LIN {X 0,Y 133.458,Z 310.494,A -85,B 0,C 180,E1 -25964.008,E2 -25964.008} C_VEL
LIN {X 0,Y 138.592,Z 326.058,A -85,B 0,C 180,E1 -25966.491,E2 -25966.491} C_VEL
LIN {X 0,Y 134.753,Z 373.673,A -85,B 0,C 180,E1 -25969.183,E2 -25969.183} C_VEL
LIN {X 0,Y 132.897,Z 387.385,A -85,B 0,C 180,E1 -25970.481,E2 -25970.481} C_VEL
LIN {X 0,Y 130.585,Z 400,A -85,B 0,C 180,E1 -25972.246,E2 -25972.246} C_VEL
LIN {X 0,Y 127.54,Z 412.416,A -85,B 0,C 180,E1 -25974.642,E2 -25974.642} C_VEL
LIN {X 0,Y 124.46,Z 423.666,A -85,B 0,C 180,E1 -25977.554,E2 -25977.554} C_VEL
LIN {X 0,Y 121.733,Z 432.92,A -85,B 0,C 180,E1 -25980.641,E2 -25980.641} C_VEL
LIN {X 0,Y 118.797,Z 442.262,A -85,B 0,C 180,E1 -25984.596,E2 -25984.596} C_VEL
LIN {X 0,Y 115.975,Z 451.38,A -85,B 0,C 180,E1 -25989.602,E2 -25989.602} C_VEL
LIN {X 0,Y 113.968,Z 458.709,A -85,B 0,C 180,E1 -25994.8,E2 -25994.8} C_VEL
LIN {X 0,Y 112.959,Z 463.637,A -85,B 0,C 180,E1 -25999.236,E2 -25999.236} C_VEL
LIN {X 0,Y 112.321,Z 468.377,A -85,B 0,C 180,E1 -26004.608,E2 -26004.608} C_VEL
LIN {X 0,Y 112.287,Z 471.952,A -85,B 0,C 180,E1 -26009.994,E2 -26009.994} C_VEL
LIN {X 0,Y 112.224,Z 473.743,A -85,B 0,C 180,E1 -26013.584,E2 -26013.584} C_VEL
LIN {X 0,Y 112.956,Z 476.023,A -85,B 0,C 180,E1 -26020.751,E2 -26020.751} C_VEL
LIN {X 0,Y 115.182,Z 476.815,A -85,B 0,C 180,E1 -26027.757,E2 -26027.757} C_VEL
LIN {X 0,Y 116.858,Z 476.66,A -85,B 0,C 180,E1 -26031.146,E2 -26031.146} C_VEL
LIN {X 0,Y 121.585,Z 475.187,A -85,B 0,C 180,E1 -26037.537,E2 -26037.537} C_VEL
LIN {X 0,Y 127.888,Z 472.229,A -85,B 0,C 180,E1 -26043.329,E2 -26043.329} C_VEL
LIN {X 0,Y 133.433,Z 468.921,A -85,B 0,C 180,E1 -26047.273,E2 -26047.273} C_VEL
LIN {X 0,Y 139.39,Z 464.647,A -85,B 0,C 180,E1 -26050.947,E2 -26050.947} C_VEL
LIN {X 0,Y 147.094,Z 458.334,A -85,B 0,C 180,E1 -26054.801,E2 -26054.801} C_VEL
LIN {X 0,Y 154.423,Z 451.461,A -85,B 0,C 180,E1 -26057.686,E2 -26057.686} C_VEL
LIN {X 0,Y 162.158,Z 442.984,A -85,B 0,C 180,E1 -26060.283,E2 -26060.283} C_VEL
LIN {X 0,Y 167.383,Z 436.409,A -85,B 0,C 180,E1 -26061.858,E2 -26061.858} C_VEL
LIN {X 0,Y 169.188,Z 433.697,A -85,B 0,C 180,E1 -26062.656,E2 -26062.656} C_VEL
LIN {X 0,Y 173.08,Z 425.278,A -85,B 0,C 180,E1 -26065.952,E2 -26065.952} C_VEL
LIN {X 0,Y 174.765,Z 422.223,A -85,B 0,C 180,E1 -26066.572,E2 -26066.572} C_VEL
LIN {X 0,Y 181.361,Z 410.201,A -85,B 0,C 180,E1 -26067.953,E2 -26067.953} C_VEL
LIN {X 0,Y 186.656,Z 398.083,A -85,B 0,C 180,E1 -26068.927,E2 -26068.927} C_VEL
LIN {X 0,Y 191.007,Z 385.003,A -85,B 0,C 180,E1 -26069.673,E2 -26069.673} C_VEL
LIN {X 0,Y 194.112,Z 371.695,A -85,B 0,C 180,E1 -26070.205,E2 -26070.205} C_VEL
LIN {X 0,Y 194.411,Z 369.647,A -85,B 0,C 180,E1 -26070.334,E2 -26070.334} C_VEL
LIN {X 0,Y 193.847,Z 366.809,A -85,B 0,C 180,E1 -26072.366,E2 -26072.366} C_VEL
LIN {X 0,Y 193.455,Z 365.322,A -85,B 0,C 180,E1 -26073.861,E2 -26073.861} C_VEL
LIN {X 0,Y 193.075,Z 363.543,A -85,B 0,C 180,E1 -26077.326,E2 -26077.326} C_VEL
LIN {X 0,Y 193.275,Z 363.614,A -85,B 0,C 180,E1 -26080.517,E2 -26080.517} C_VEL
LIN {X 0,Y 194.066,Z 365.581,A -85,B 0,C 180,E1 -26083.959,E2 -26083.959} C_VEL
LIN {X 0,Y 194.678,Z 367.91,A -85,B 0,C 180,E1 -26085.889,E2 -26085.889} C_VEL
LIN {X 0,Y 191.67,Z 382.126,A -85,B 0,C 180,E1 -26086.438,E2 -26086.438} C_VEL
LIN {X 0,Y 187.36,Z 395.537,A -85,B 0,C 180,E1 -26087.213,E2 -26087.213} C_VEL
LIN {X 0,Y 182.064,Z 408.153,A -85,B 0,C 180,E1 -26088.293,E2 -26088.293} C_VEL
LIN {X 0,Y 175.888,Z 419.646,A -85,B 0,C 180,E1 -26089.63,E2 -26089.63} C_VEL
LIN {X 0,Y 168.761,Z 430.521,A -85,B 0,C 180,E1 -26091.34,E2 -26091.34} C_VEL
LIN {X 0,Y 161.795,Z 439.402,A -85,B 0,C 180,E1 -26093.213,E2 -26093.213} C_VEL
LIN {X 0,Y 154.101,Z 447.705,A -85,B 0,C 180,E1 -26095.585,E2 -26095.585} C_VEL
LIN {X 0,Y 145.288,Z 455.81,A -85,B 0,C 180,E1 -26098.796,E2 -26098.796} C_VEL
LIN {X 0,Y 138.496,Z 461.105,A -85,B 0,C 180,E1 -26101.734,E2 -26101.734} C_VEL
LIN {X 0,Y 132.107,Z 465.384,A -85,B 0,C 180,E1 -26104.966,E2 -26104.966} C_VEL
LIN {X 0,Y 124.615,Z 469.621,A -85,B 0,C 180,E1 -26109.719,E2 -26109.719} C_VEL
LIN {X 0,Y 119.758,Z 471.813,A -85,B 0,C 180,E1 -26113.553,E2 -26113.553} C_VEL
LIN {X 0,Y 115.476,Z 473.325,A -85,B 0,C 180,E1 -26117.691,E2 -26117.691} C_VEL
LIN {X 0,Y 111.912,Z 474.12,A -85,B 0,C 180,E1 -26122.108,E2 -26122.108} C_VEL
LIN {X 0,Y 109.007,Z 474.248,A -85,B 0,C 180,E1 -26126.799,E2 -26126.799} C_VEL
LIN {X 0,Y 106.871,Z 473.73,A -85,B 0,C 180,E1 -26131.71,E2 -26131.71} C_VEL
LIN {X 0,Y 104.955,Z 471.543,A -85,B 0,C 180,E1 -26139.466,E2 -26139.466} C_VEL
LIN {X 0,Y 104.493,Z 468.971,A -85,B 0,C 180,E1 -26145.085,E2 -26145.085} C_VEL
LIN {X 0,Y 104.749,Z 465.683,A -85,B 0,C 180,E1 -26150.412,E2 -26150.412} C_VEL
LIN {X 0,Y 105.789,Z 460.351,A -85,B 0,C 180,E1 -26156.838,E2 -26156.838} C_VEL
LIN {X 0,Y 107.416,Z 453.895,A -85,B 0,C 180,E1 -26162.75,E2 -26162.75} C_VEL
LIN {X 0,Y 109.827,Z 445.968,A -85,B 0,C 180,E1 -26168.341,E2 -26168.341} C_VEL
LIN {X 0,Y 112.799,Z 436.816,A -85,B 0,C 180,E1 -26173.259,E2 -26173.259} C_VEL
LIN {X 0,Y 115.9,Z 427.136,A -85,B 0,C 180,E1 -26177.297,E2 -26177.297} C_VEL
LIN {X 0,Y 119.13,Z 416.62,A -85,B 0,C 180,E1 -26180.684,E2 -26180.684} C_VEL
LIN {X 0,Y 122.359,Z 404.541,A -85,B 0,C 180,E1 -26183.616,E2 -26183.616} C_VEL
LIN {X 0,Y 125.028,Z 392.632,A -85,B 0,C 180,E1 -26185.775,E2 -26185.775} C_VEL
LIN {X 0,Y 127.359,Z 379.198,A -85,B 0,C 180,E1 -26187.493,E2 -26187.493} C_VEL
LIN {X 0,Y 129.121,Z 364.891,A -85,B 0,C 180,E1 -26188.636,E2 -26188.636} C_VEL
LIN {X 0,Y 132.327,Z 323.972,A -85,B 0,C 180,E1 -26191.019,E2 -26191.019} C_VEL
LIN {X 0,Y 127.72,Z 309.873,A -85,B 0,C 180,E1 -26193.47,E2 -26193.47} C_VEL
LIN {X 0,Y 120.856,Z 294.809,A -85,B 0,C 180,E1 -26196.985,E2 -26196.985} C_VEL
LIN {X 0,Y 112.645,Z 281.335,A -85,B 0,C 180,E1 -26201.497,E2 -26201.497} C_VEL
LIN {X 0,Y 110.503,Z 277.97,A -85,B 0,C 180,E1 -26202.824,E2 -26202.824} C_VEL
LIN {X 0,Y 108.695,Z 275.672,A -85,B 0,C 180,E1 -26203.912,E2 -26203.912} C_VEL
LIN {X 0,Y 108.069,Z 274.008,A -85,B 0,C 180,E1 -26204.766,E2 -26204.766} C_VEL
LIN {X 0,Y 107.913,Z 273.542,A -85,B 0,C 180,E1 -26206.075,E2 -26206.075} C_VEL
LIN {X 0,Y 107.862,Z 273.55,A -85,B 0,C 180,E1 -26213.02,E2 -26213.02} C_VEL
LIN {X 0,Y 107.766,Z 273.521,A -85,B 0,C 180,E1 -26221.455,E2 -26221.455} C_VEL
LIN {X 0,Y 107.72,Z 273.55,A -85,B 0,C 180,E1 -26228.516,E2 -26228.516} C_VEL
LIN {X 0,Y 107.752,Z 273.545,A -85,B 0,C 180,E1 -26235.854,E2 -26235.854} C_VEL
LIN {X 0,Y 107.768,Z 273.559,A -85,B 0,C 180,E1 -26241.506,E2 -26241.506} C_VEL
LIN {X 0,Y 107.79,Z 273.555,A -85,B 0,C 180,E1 -26248.591,E2 -26248.591} C_VEL
LIN {X 0,Y 107.877,Z 273.535,A -85,B 0,C 180,E1 -26257.019,E2 -26257.019} C_VEL
LIN {X 0,Y 107.967,Z 273.514,A -85,B 0,C 180,E1 -26264.934,E2 -26264.934} C_VEL
LIN {X 0,Y 108.225,Z 273.503,A -85,B 0,C 180,E1 -26268.792,E2 -26268.792} C_VEL
LIN {X 0,Y 108.292,Z 273.473,A -85,B 0,C 180,E1 -26272.567,E2 -26272.567} C_VEL
LIN {X 0,Y 108.906,Z 273.401,A -85,B 0,C 180,E1 -26280.024,E2 -26280.024} C_VEL
LIN {X 0,Y 108.3,Z 273.432,A -85,B 0,C 180,E1 -26287.481,E2 -26287.481} C_VEL
LIN {X 0,Y 108.158,Z 273.513,A -85,B 0,C 180,E1 -26292.894,E2 -26292.894} C_VEL
LIN {X 0,Y 107.889,Z 273.496,A -85,B 0,C 180,E1 -26299.033,E2 -26299.033} C_VEL
LIN {X 0,Y 107.862,Z 273.551,A -85,B 0,C 180,E1 -26304.175,E2 -26304.175} C_VEL
LIN {X 0,Y 107.867,Z 273.734,A -85,B 0,C 180,E1 -26310.625,E2 -26310.625} C_VEL
LIN {X 0,Y 108.13,Z 274.915,A -85,B 0,C 180,E1 -26311.483,E2 -26311.483} C_VEL
LIN {X 0,Y 109.862,Z 277.767,A -85,B 0,C 180,E1 -26312.662,E2 -26312.662} C_VEL
LIN {X 0,Y 110.865,Z 279.219,A -85,B 0,C 180,E1 -26313.266,E2 -26313.266} C_VEL
LIN {X 0,Y 115.315,Z 286.508,A -85,B 0,C 180,E1 -26315.915,E2 -26315.915} C_VEL
LIN {X 0,Y 122.163,Z 298.987,A -85,B 0,C 180,E1 -26319.617,E2 -26319.617} C_VEL
LIN {X 0,Y 125.721,Z 307.389,A -85,B 0,C 180,E1 -26321.483,E2 -26321.483} C_VEL
LIN {X 0,Y 131.917,Z 326.077,A -85,B 0,C 180,E1 -26324.815,E2 -26324.815} C_VEL
LIN {X 0,Y 132.361,Z 327.576,A -85,B 0,C 180,E1 -26325.05,E2 -26325.05} C_VEL
LIN {X 0,Y 128.534,Z 373.038,A -85,B 0,C 180,E1 -26327.698,E2 -26327.698} C_VEL
LIN {X 0,Y 126.628,Z 386.825,A -85,B 0,C 180,E1 -26329.028,E2 -26329.028} C_VEL
LIN {X 0,Y 124.096,Z 400.074,A -85,B 0,C 180,E1 -26330.94,E2 -26330.94} C_VEL
LIN {X 0,Y 120.949,Z 412.457,A -85,B 0,C 180,E1 -26333.438,E2 -26333.438} C_VEL
LIN {X 0,Y 117.615,Z 424.174,A -85,B 0,C 180,E1 -26336.634,E2 -26336.634} C_VEL
LIN {X 0,Y 114.218,Z 434.841,A -85,B 0,C 180,E1 -26340.505,E2 -26340.505} C_VEL
LIN {X 0,Y 111.279,Z 443.885,A -85,B 0,C 180,E1 -26344.76,E2 -26344.76} C_VEL
LIN {X 0,Y 108.457,Z 452.691,A -85,B 0,C 180,E1 -26350.105,E2 -26350.105} C_VEL
LIN {X 0,Y 106.605,Z 459.7,A -85,B 0,C 180,E1 -26355.68,E2 -26355.68} C_VEL
LIN {X 0,Y 105.434,Z 466.068,A -85,B 0,C 180,E1 -26362.332,E2 -26362.332} C_VEL
LIN {X 0,Y 105.165,Z 470.184,A -85,B 0,C 180,E1 -26368.079,E2 -26368.079} C_VEL
LIN {X 0,Y 105.172,Z 473.18,A -85,B 0,C 180,E1 -26373.825,E2 -26373.825} C_VEL
LIN {X 0,Y 105.99,Z 475.711,A -85,B 0,C 180,E1 -26381.467,E2 -26381.467} C_VEL
LIN {X 0,Y 108.434,Z 476.672,A -85,B 0,C 180,E1 -26388.902,E2 -26388.902} C_VEL
LIN {X 0,Y 112.569,Z 476.193,A -85,B 0,C 180,E1 -26395.907,E2 -26395.907} C_VEL
LIN {X 0,Y 115.342,Z 475.403,A -85,B 0,C 180,E1 -26399.166,E2 -26399.166} C_VEL
LIN {X 0,Y 122.024,Z 472.634,A -85,B 0,C 180,E1 -26405.159,E2 -26405.159} C_VEL
LIN {X 0,Y 129.85,Z 468.328,A -85,B 0,C 180,E1 -26410.495,E2 -26410.495} C_VEL
LIN {X 0,Y 136.402,Z 463.94,A -85,B 0,C 180,E1 -26414.065,E2 -26414.065} C_VEL
LIN {X 0,Y 144.716,Z 457.406,A -85,B 0,C 180,E1 -26417.775,E2 -26417.775} C_VEL
LIN {X 0,Y 153.762,Z 449.031,A -85,B 0,C 180,E1 -26420.98,E2 -26420.98} C_VEL
LIN {X 0,Y 161.929,Z 440.115,A -85,B 0,C 180,E1 -26423.403,E2 -26423.403} C_VEL
LIN {X 0,Y 169.65,Z 430.011,A -85,B 0,C 180,E1 -26425.413,E2 -26425.413} C_VEL
LIN {X 0,Y 174.765,Z 422.223,A -85,B 0,C 180,E1 -26426.572,E2 -26426.572} C_VEL
LIN {X 0,Y 176.699,Z 418.614,A -85,B 0,C 180,E1 -26427.301,E2 -26427.301} C_VEL
LIN {X 0,Y 180.282,Z 409.617,A -85,B 0,C 180,E1 -26430.024,E2 -26430.024} C_VEL
LIN {X 0,Y 181.764,Z 406.275,A -85,B 0,C 180,E1 -26430.514,E2 -26430.514} C_VEL
LIN {X 0,Y 186.652,Z 394.633,A -85,B 0,C 180,E1 -26431.305,E2 -26431.305} C_VEL
LIN {X 0,Y 190.694,Z 381.847,A -85,B 0,C 180,E1 -26431.916,E2 -26431.916} C_VEL
LIN {X 0,Y 192.442,Z 374.289,A -85,B 0,C 180,E1 -26432.244,E2 -26432.244} C_VEL
LIN {X 0,Y 192.117,Z 372.167,A -85,B 0,C 180,E1 -26434.26,E2 -26434.26} C_VEL
LIN {X 0,Y 191.881,Z 370.577,A -85,B 0,C 180,E1 -26437.177,E2 -26437.177} C_VEL
LIN {X 0,Y 192.052,Z 370.646,A -85,B 0,C 180,E1 -26440.469,E2 -26440.469} C_VEL
LIN {X 0,Y 192.619,Z 372.555,A -85,B 0,C 180,E1 -26443.667,E2 -26443.667} C_VEL
LIN {X 0,Y 192.681,Z 372.889,A -85,B 0,C 180,E1 -26443.967,E2 -26443.967} C_VEL
LIN {X 0,Y 189.302,Z 386.287,A -85,B 0,C 180,E1 -26444.523,E2 -26444.523} C_VEL
LIN {X 0,Y 185.011,Z 398.447,A -85,B 0,C 180,E1 -26445.258,E2 -26445.258} C_VEL
LIN {X 0,Y 179.842,Z 409.73,A -85,B 0,C 180,E1 -26446.216,E2 -26446.216} C_VEL
LIN {X 0,Y 173.57,Z 420.765,A -85,B 0,C 180,E1 -26447.469,E2 -26447.469} C_VEL
LIN {X 0,Y 166.417,Z 431.16,A -85,B 0,C 180,E1 -26449.049,E2 -26449.049} C_VEL
LIN {X 0,Y 159.291,Z 439.856,A -85,B 0,C 180,E1 -26450.814,E2 -26450.814} C_VEL
LIN {X 0,Y 151.423,Z 447.995,A -85,B 0,C 180,E1 -26453.055,E2 -26453.055} C_VEL
LIN {X 0,Y 142.266,Z 455.957,A -85,B 0,C 180,E1 -26456.106,E2 -26456.106} C_VEL
LIN {X 0,Y 133.52,Z 462.291,A -85,B 0,C 180,E1 -26459.655,E2 -26459.655} C_VEL
LIN {X 0,Y 126.358,Z 466.639,A -85,B 0,C 180,E1 -26463.167,E2 -26463.167} C_VEL
LIN {X 0,Y 117.802,Z 470.811,A -85,B 0,C 180,E1 -26468.553,E2 -26468.553} C_VEL
LIN {X 0,Y 110.463,Z 473.381,A -85,B 0,C 180,E1 -26474.718,E2 -26474.718} C_VEL
LIN {X 0,Y 105.25,Z 474.34,A -85,B 0,C 180,E1 -26480.818,E2 -26480.818} C_VEL
LIN {X 0,Y 101.901,Z 474.258,A -85,B 0,C 180,E1 -26486.303,E2 -26486.303} C_VEL
LIN {X 0,Y 98.767,Z 472.67,A -85,B 0,C 180,E1 -26494.663,E2 -26494.663} C_VEL
LIN {X 0,Y 97.732,Z 470.74,A -85,B 0,C 180,E1 -26500.292,E2 -26500.292} C_VEL
LIN {X 0,Y 97.497,Z 466.872,A -85,B 0,C 180,E1 -26507.895,E2 -26507.895} C_VEL
LIN {X 0,Y 98.095,Z 462.882,A -85,B 0,C 180,E1 -26513.647,E2 -26513.647} C_VEL
LIN {X 0,Y 99.518,Z 456.76,A -85,B 0,C 180,E1 -26520.382,E2 -26520.382} C_VEL
LIN {X 0,Y 101.733,Z 449.333,A -85,B 0,C 180,E1 -26526.603,E2 -26526.603} C_VEL
LIN {X 0,Y 104.335,Z 441.294,A -85,B 0,C 180,E1 -26531.779,E2 -26531.779} C_VEL
LIN {X 0,Y 107.743,Z 431.313,A -85,B 0,C 180,E1 -26536.731,E2 -26536.731} C_VEL
LIN {X 0,Y 110.996,Z 421.556,A -85,B 0,C 180,E1 -26540.44,E2 -26540.44} C_VEL
LIN {X 0,Y 114.565,Z 409.698,A -85,B 0,C 180,E1 -26543.843,E2 -26543.843} C_VEL
LIN {X 0,Y 117.808,Z 396.842,A -85,B 0,C 180,E1 -26546.586,E2 -26546.586} C_VEL
LIN {X 0,Y 120.363,Z 383.935,A -85,B 0,C 180,E1 -26548.523,E2 -26548.523} C_VEL
LIN {X 0,Y 122.302,Z 371.003,A -85,B 0,C 180,E1 -26549.823,E2 -26549.823} C_VEL
LIN {X 0,Y 126.249,Z 325.619,A -85,B 0,C 180,E1 -26552.595,E2 -26552.595} C_VEL
LIN {X 0,Y 122.186,Z 313.065,A -85,B 0,C 180,E1 -26554.915,E2 -26554.915} C_VEL
LIN {X 0,Y 115.891,Z 298.992,A -85,B 0,C 180,E1 -26558.409,E2 -26558.409} C_VEL
LIN {X 0,Y 108.378,Z 286.324,A -85,B 0,C 180,E1 -26562.891,E2 -26562.891} C_VEL
LIN {X 0,Y 105.892,Z 282.719,A -85,B 0,C 180,E1 -26564.475,E2 -26564.475} C_VEL
LIN {X 0,Y 103.327,Z 278.957,A -85,B 0,C 180,E1 -26566.224,E2 -26566.224} C_VEL
LIN {X 0,Y 101.368,Z 276.297,A -85,B 0,C 180,E1 -26567.667,E2 -26567.667} C_VEL
LIN {X 0,Y 100.904,Z 274.916,A -85,B 0,C 180,E1 -26568.537,E2 -26568.537} C_VEL
LIN {X 0,Y 100.798,Z 274.481,A -85,B 0,C 180,E1 -26569.349,E2 -26569.349} C_VEL
LIN {X 0,Y 100.732,Z 274.41,A -85,B 0,C 180,E1 -26574.977,E2 -26574.977} C_VEL
LIN {X 0,Y 100.667,Z 274.425,A -85,B 0,C 180,E1 -26583.149,E2 -26583.149} C_VEL
LIN {X 0,Y 100.669,Z 274.43,A -85,B 0,C 180,E1 -26589.876,E2 -26589.876} C_VEL
LIN {X 0,Y 100.716,Z 274.42,A -85,B 0,C 180,E1 -26595.79,E2 -26595.79} C_VEL
LIN {X 0,Y 100.707,Z 274.44,A -85,B 0,C 180,E1 -26601.128,E2 -26601.128} C_VEL
LIN {X 0,Y 100.691,Z 274.424,A -85,B 0,C 180,E1 -26606.895,E2 -26606.895} C_VEL
LIN {X 0,Y 100.733,Z 274.414,A -85,B 0,C 180,E1 -26615.284,E2 -26615.284} C_VEL
LIN {X 0,Y 100.779,Z 274.431,A -85,B 0,C 180,E1 -26619.623,E2 -26619.623} C_VEL
LIN {X 0,Y 101.124,Z 274.387,A -85,B 0,C 180,E1 -26627.993,E2 -26627.993} C_VEL
LIN {X 0,Y 101.228,Z 274.354,A -85,B 0,C 180,E1 -26632.045,E2 -26632.045} C_VEL
LIN {X 0,Y 101.834,Z 274.279,A -85,B 0,C 180,E1 -26640.026,E2 -26640.026} C_VEL
LIN {X 0,Y 101.238,Z 274.314,A -85,B 0,C 180,E1 -26648.007,E2 -26648.007} C_VEL
LIN {X 0,Y 101.071,Z 274.394,A -85,B 0,C 180,E1 -26653.195,E2 -26653.195} C_VEL
LIN {X 0,Y 100.811,Z 274.382,A -85,B 0,C 180,E1 -26660.427,E2 -26660.427} C_VEL
LIN {X 0,Y 100.737,Z 274.597,A -85,B 0,C 180,E1 -26666.77,E2 -26666.77} C_VEL
LIN {X 0,Y 101.026,Z 275.692,A -85,B 0,C 180,E1 -26667.766,E2 -26667.766} C_VEL
LIN {X 0,Y 102.613,Z 278.345,A -85,B 0,C 180,E1 -26669.096,E2 -26669.096} C_VEL
LIN {X 0,Y 103.732,Z 279.708,A -85,B 0,C 180,E1 -26669.865,E2 -26669.865} C_VEL
LIN {X 0,Y 105.926,Z 283.137,A -85,B 0,C 180,E1 -26671.387,E2 -26671.387} C_VEL
LIN {X 0,Y 111.251,Z 292.064,A -85,B 0,C 180,E1 -26674.772,E2 -26674.772} C_VEL
LIN {X 0,Y 117.626,Z 304.047,A -85,B 0,C 180,E1 -26678.494,E2 -26678.494} C_VEL
LIN {X 0,Y 121.537,Z 314.302,A -85,B 0,C 180,E1 -26680.763,E2 -26680.763} C_VEL
LIN {X 0,Y 126.17,Z 328.859,A -85,B 0,C 180,E1 -26683.434,E2 -26683.434} C_VEL
LIN {X 0,Y 122.853,Z 368.787,A -85,B 0,C 180,E1 -26685.845,E2 -26685.845} C_VEL
LIN {X 0,Y 121.12,Z 382.525,A -85,B 0,C 180,E1 -26687.009,E2 -26687.009} C_VEL
LIN {X 0,Y 118.853,Z 394.699,A -85,B 0,C 180,E1 -26688.576,E2 -26688.576} C_VEL
LIN {X 0,Y 116.251,Z 405.845,A -85,B 0,C 180,E1 -26690.589,E2 -26690.589} C_VEL
LIN {X 0,Y 113.144,Z 416.972,A -85,B 0,C 180,E1 -26693.276,E2 -26693.276} C_VEL
LIN {X 0,Y 109.613,Z 428.253,A -85,B 0,C 180,E1 -26696.887,E2 -26696.887} C_VEL
LIN {X 0,Y 106.104,Z 438.602,A -85,B 0,C 180,E1 -26701.294,E2 -26701.294} C_VEL
LIN {X 0,Y 102.748,Z 448.422,A -85,B 0,C 180,E1 -26706.833,E2 -26706.833} C_VEL
LIN {X 0,Y 100.314,Z 456.252,A -85,B 0,C 180,E1 -26712.67,E2 -26712.67} C_VEL
LIN {X 0,Y 99.035,Z 461.585,A -85,B 0,C 180,E1 -26717.701,E2 -26717.701} C_VEL
LIN {X 0,Y 98.23,Z 466.709,A -85,B 0,C 180,E1 -26723.832,E2 -26723.832} C_VEL
LIN {X 0,Y 98.154,Z 470.641,A -85,B 0,C 180,E1 -26729.993,E2 -26729.993} C_VEL
LIN {X 0,Y 98.102,Z 472.61,A -85,B 0,C 180,E1 -26734.101,E2 -26734.101} C_VEL
LIN {X 0,Y 99.051,Z 475.333,A -85,B 0,C 180,E1 -26742.283,E2 -26742.283} C_VEL
LIN {X 0,Y 101.72,Z 476.525,A -85,B 0,C 180,E1 -26750.202,E2 -26750.202} C_VEL
LIN {X 0,Y 106.234,Z 476.23,A -85,B 0,C 180,E1 -26757.579,E2 -26757.579} C_VEL
LIN {X 0,Y 112.582,Z 474.499,A -85,B 0,C 180,E1 -26764.175,E2 -26764.175} C_VEL
LIN {X 0,Y 116.296,Z 473.066,A -85,B 0,C 180,E1 -26767.172,E2 -26767.172} C_VEL
LIN {X 0,Y 124.568,Z 468.985,A -85,B 0,C 180,E1 -26772.603,E2 -26772.603} C_VEL
LIN {X 0,Y 131.444,Z 464.813,A -85,B 0,C 180,E1 -26776.196,E2 -26776.196} C_VEL
LIN {X 0,Y 138.807,Z 459.589,A -85,B 0,C 180,E1 -26779.409,E2 -26779.409} C_VEL
LIN {X 0,Y 148.112,Z 451.932,A -85,B 0,C 180,E1 -26782.628,E2 -26782.628} C_VEL
LIN {X 0,Y 156.501,Z 443.669,A -85,B 0,C 180,E1 -26785.031,E2 -26785.031} C_VEL
LIN {X 0,Y 163.656,Z 435.338,A -85,B 0,C 180,E1 -26786.858,E2 -26786.858} C_VEL
LIN {X 0,Y 171.046,Z 425.212,A -85,B 0,C 180,E1 -26788.485,E2 -26788.485} C_VEL
LIN {X 0,Y 177.834,Z 414.057,A -85,B 0,C 180,E1 -26789.816,E2 -26789.816} C_VEL
LIN {X 0,Y 181.764,Z 406.275,A -85,B 0,C 180,E1 -26790.514,E2 -26790.514} C_VEL
LIN {X 0,Y 183.237,Z 402.856,A -85,B 0,C 180,E1 -26790.973,E2 -26790.973} C_VEL
LIN {X 0,Y 186.584,Z 392.322,A -85,B 0,C 180,E1 -26793.388,E2 -26793.388} C_VEL
LIN {X 0,Y 187.728,Z 388.725,A -85,B 0,C 180,E1 -26793.769,E2 -26793.769} C_VEL
LIN {X 0,Y 190.429,Z 379.365,A -85,B 0,C 180,E1 -26794.188,E2 -26794.188} C_VEL
LIN {X 0,Y 190.352,Z 377.481,A -85,B 0,C 180,E1 -26797.361,E2 -26797.361} C_VEL
LIN {X 0,Y 190.49,Z 377.553,A -85,B 0,C 180,E1 -26800.302,E2 -26800.302} C_VEL
LIN {X 0,Y 190.622,Z 378.43,A -85,B 0,C 180,E1 -26802.035,E2 -26802.035} C_VEL
LIN {X 0,Y 186.901,Z 390.853,A -85,B 0,C 180,E1 -26802.62,E2 -26802.62} C_VEL
LIN {X 0,Y 182.801,Z 401.272,A -85,B 0,C 180,E1 -26803.261,E2 -26803.261} C_VEL
LIN {X 0,Y 177.365,Z 412.324,A -85,B 0,C 180,E1 -26804.177,E2 -26804.177} C_VEL
LIN {X 0,Y 171.288,Z 422.4,A -85,B 0,C 180,E1 -26805.3,E2 -26805.3} C_VEL
LIN {X 0,Y 164.238,Z 432.078,A -85,B 0,C 180,E1 -26806.725,E2 -26806.725} C_VEL
LIN {X 0,Y 155.854,Z 441.649,A -85,B 0,C 180,E1 -26808.639,E2 -26808.639} C_VEL
LIN {X 0,Y 146.266,Z 450.772,A -85,B 0,C 180,E1 -26811.212,E2 -26811.212} C_VEL
LIN {X 0,Y 137.314,Z 457.826,A -85,B 0,C 180,E1 -26814.106,E2 -26814.106} C_VEL
LIN {X 0,Y 128.246,Z 463.749,A -85,B 0,C 180,E1 -26817.626,E2 -26817.626} C_VEL
LIN {X 0,Y 119.525,Z 468.39,A -85,B 0,C 180,E1 -26821.856,E2 -26821.856} C_VEL
LIN {X 0,Y 111.018,Z 471.874,A -85,B 0,C 180,E1 -26827.249,E2 -26827.249} C_VEL
LIN {X 0,Y 105.787,Z 473.451,A -85,B 0,C 180,E1 -26831.47,E2 -26831.47} C_VEL
LIN {X 0,Y 101.225,Z 474.291,A -85,B 0,C 180,E1 -26836.096,E2 -26836.096} C_VEL
LIN {X 0,Y 97.459,Z 474.5,A -85,B 0,C 180,E1 -26841.104,E2 -26841.104} C_VEL
LIN {X 0,Y 94.354,Z 474.009,A -85,B 0,C 180,E1 -26846.66,E2 -26846.66} C_VEL
LIN {X 0,Y 92.073,Z 472.679,A -85,B 0,C 180,E1 -26852.913,E2 -26852.913} C_VEL
LIN {X 0,Y 90.757,Z 470.563,A -85,B 0,C 180,E1 -26859.264,E2 -26859.264} C_VEL
LIN {X 0,Y 90.323,Z 467.669,A -85,B 0,C 180,E1 -26865.562,E2 -26865.562} C_VEL
LIN {X 0,Y 90.729,Z 463.961,A -85,B 0,C 180,E1 -26871.717,E2 -26871.717} C_VEL
LIN {X 0,Y 92.027,Z 458.157,A -85,B 0,C 180,E1 -26878.979,E2 -26878.979} C_VEL
LIN {X 0,Y 94.084,Z 451.007,A -85,B 0,C 180,E1 -26885.75,E2 -26885.75} C_VEL
LIN {X 0,Y 96.514,Z 443.731,A -85,B 0,C 180,E1 -26891.102,E2 -26891.102} C_VEL
LIN {X 0,Y 99.711,Z 434.91,A -85,B 0,C 180,E1 -26896.164,E2 -26896.164} C_VEL
LIN {X 0,Y 103.326,Z 424.481,A -85,B 0,C 180,E1 -26900.71,E2 -26900.71} C_VEL
LIN {X 0,Y 107.028,Z 413.26,A -85,B 0,C 180,E1 -26904.379,E2 -26904.379} C_VEL
LIN {X 0,Y 110.026,Z 402.582,A -85,B 0,C 180,E1 -26907.041,E2 -26907.041} C_VEL
LIN {X 0,Y 112.99,Z 390.041,A -85,B 0,C 180,E1 -26909.323,E2 -26909.323} C_VEL
LIN {X 0,Y 115.381,Z 376.362,A -85,B 0,C 180,E1 -26911.068,E2 -26911.068} C_VEL
LIN {X 0,Y 117.09,Z 362.692,A -85,B 0,C 180,E1 -26912.098,E2 -26912.098} C_VEL
LIN {X 0,Y 120.204,Z 327.274,A -85,B 0,C 180,E1 -26914.286,E2 -26914.286} C_VEL
LIN {X 0,Y 116.812,Z 316.497,A -85,B 0,C 180,E1 -26916.41,E2 -26916.41} C_VEL
LIN {X 0,Y 111.022,Z 303.213,A -85,B 0,C 180,E1 -26919.946,E2 -26919.946} C_VEL
LIN {X 0,Y 103.743,Z 290.76,A -85,B 0,C 180,E1 -26924.63,E2 -26924.63} C_VEL
LIN {X 0,Y 101.563,Z 287.576,A -85,B 0,C 180,E1 -26926.145,E2 -26926.145} C_VEL
LIN {X 0,Y 99.14,Z 284.009,A -85,B 0,C 180,E1 -26927.962,E2 -26927.962} C_VEL
LIN {X 0,Y 96.507,Z 280.107,A -85,B 0,C 180,E1 -26930.118,E2 -26930.118} C_VEL
LIN {X 0,Y 94.381,Z 277.664,A -85,B 0,C 180,E1 -26931.917,E2 -26931.917} C_VEL
LIN {X 0,Y 93.761,Z 275.909,A -85,B 0,C 180,E1 -26932.947,E2 -26932.947} C_VEL
LIN {X 0,Y 93.677,Z 275.366,A -85,B 0,C 180,E1 -26933.905,E2 -26933.905} C_VEL
LIN {X 0,Y 93.549,Z 275.29,A -85,B 0,C 180,E1 -26941.736,E2 -26941.736} C_VEL
LIN {X 0,Y 93.53,Z 275.323,A -85,B 0,C 180,E1 -26946.96,E2 -26946.96} C_VEL
LIN {X 0,Y 93.605,Z 275.326,A -85,B 0,C 180,E1 -26952.52,E2 -26952.52} C_VEL
LIN {X 0,Y 93.621,Z 275.308,A -85,B 0,C 180,E1 -26958.66,E2 -26958.66} C_VEL
LIN {X 0,Y 93.604,Z 275.302,A -85,B 0,C 180,E1 -26965.692,E2 -26965.692} C_VEL
LIN {X 0,Y 93.633,Z 275.297,A -85,B 0,C 180,E1 -26974.266,E2 -26974.266} C_VEL
LIN {X 0,Y 93.65,Z 275.314,A -85,B 0,C 180,E1 -26977.994,E2 -26977.994} C_VEL
LIN {X 0,Y 94.015,Z 275.265,A -85,B 0,C 180,E1 -26987.07,E2 -26987.07} C_VEL
LIN {X 0,Y 94.14,Z 275.239,A -85,B 0,C 180,E1 -26991.442,E2 -26991.442} C_VEL
LIN {X 0,Y 94.763,Z 275.154,A -85,B 0,C 180,E1 -27000.028,E2 -27000.028} C_VEL
LIN {X 0,Y 94.151,Z 275.2,A -85,B 0,C 180,E1 -27008.614,E2 -27008.614} C_VEL
LIN {X 0,Y 93.98,Z 275.272,A -85,B 0,C 180,E1 -27013.522,E2 -27013.522} C_VEL
LIN {X 0,Y 93.712,Z 275.367,A -85,B 0,C 180,E1 -27021.907,E2 -27021.907} C_VEL
LIN {X 0,Y 93.913,Z 276.359,A -85,B 0,C 180,E1 -27023.238,E2 -27023.238} C_VEL
LIN {X 0,Y 95.44,Z 279.088,A -85,B 0,C 180,E1 -27024.788,E2 -27024.788} C_VEL
LIN {X 0,Y 97.021,Z 280.85,A -85,B 0,C 180,E1 -27026.07,E2 -27026.07} C_VEL
LIN {X 0,Y 99.076,Z 284.025,A -85,B 0,C 180,E1 -27027.771,E2 -27027.771} C_VEL
LIN {X 0,Y 104.452,Z 292.648,A -85,B 0,C 180,E1 -27031.74,E2 -27031.74} C_VEL
LIN {X 0,Y 110.497,Z 303.838,A -85,B 0,C 180,E1 -27035.673,E2 -27035.673} C_VEL
LIN {X 0,Y 113.815,Z 310.987,A -85,B 0,C 180,E1 -27037.738,E2 -27037.738} C_VEL
LIN {X 0,Y 118.513,Z 325.074,A -85,B 0,C 180,E1 -27040.742,E2 -27040.742} C_VEL
LIN {X 0,Y 120.169,Z 330.598,A -85,B 0,C 180,E1 -27041.771,E2 -27041.771} C_VEL
LIN {X 0,Y 116.09,Z 373.993,A -85,B 0,C 180,E1 -27044.494,E2 -27044.494} C_VEL
LIN {X 0,Y 114.124,Z 386.748,A -85,B 0,C 180,E1 -27045.834,E2 -27045.834} C_VEL
LIN {X 0,Y 111.377,Z 399.93,A -85,B 0,C 180,E1 -27047.891,E2 -27047.891} C_VEL
LIN {X 0,Y 107.948,Z 412.253,A -85,B 0,C 180,E1 -27050.589,E2 -27050.589} C_VEL
LIN {X 0,Y 104.694,Z 422.762,A -85,B 0,C 180,E1 -27053.701,E2 -27053.701} C_VEL
LIN {X 0,Y 100.934,Z 433.601,A -85,B 0,C 180,E1 -27057.924,E2 -27057.924} C_VEL
LIN {X 0,Y 97.359,Z 443.611,A -85,B 0,C 180,E1 -27063.174,E2 -27063.174} C_VEL
LIN {X 0,Y 94.307,Z 452.408,A -85,B 0,C 180,E1 -27069.261,E2 -27069.261} C_VEL
LIN {X 0,Y 92.35,Z 459.414,A -85,B 0,C 180,E1 -27075.673,E2 -27075.673} C_VEL
LIN {X 0,Y 91.201,Z 465.789,A -85,B 0,C 180,E1 -27083.355,E2 -27083.355} C_VEL
LIN {X 0,Y 91.079,Z 469.897,A -85,B 0,C 180,E1 -27089.992,E2 -27089.992} C_VEL
LIN {X 0,Y 91.05,Z 472.009,A -85,B 0,C 180,E1 -27094.419,E2 -27094.419} C_VEL
LIN {X 0,Y 92.117,Z 474.91,A -85,B 0,C 180,E1 -27103.223,E2 -27103.223} C_VEL
LIN {X 0,Y 95.073,Z 476.323,A -85,B 0,C 180,E1 -27111.683,E2 -27111.683} C_VEL
LIN {X 0,Y 97.227,Z 476.488,A -85,B 0,C 180,E1 -27115.695,E2 -27115.695} C_VEL
LIN {X 0,Y 103.194,Z 475.687,A -85,B 0,C 180,E1 -27123.005,E2 -27123.005} C_VEL
LIN {X 0,Y 110.726,Z 473.435,A -85,B 0,C 180,E1 -27129.39,E2 -27129.39} C_VEL
LIN {X 0,Y 117.228,Z 470.723,A -85,B 0,C 180,E1 -27133.577,E2 -27133.577} C_VEL
LIN {X 0,Y 124.228,Z 467.121,A -85,B 0,C 180,E1 -27137.336,E2 -27137.336} C_VEL
LIN {X 0,Y 131.743,Z 462.531,A -85,B 0,C 180,E1 -27140.662,E2 -27140.662} C_VEL
LIN {X 0,Y 141.205,Z 455.693,A -85,B 0,C 180,E1 -27143.968,E2 -27143.968} C_VEL
LIN {X 0,Y 149.731,Z 448.351,A -85,B 0,C 180,E1 -27146.413,E2 -27146.413} C_VEL
LIN {X 0,Y 158.513,Z 439.365,A -85,B 0,C 180,E1 -27148.584,E2 -27148.584} C_VEL
LIN {X 0,Y 166.789,Z 429.207,A -85,B 0,C 180,E1 -27150.342,E2 -27150.342} C_VEL
LIN {X 0,Y 173.754,Z 418.951,A -85,B 0,C 180,E1 -27151.602,E2 -27151.602} C_VEL
LIN {X 0,Y 179.986,Z 407.638,A -85,B 0,C 180,E1 -27152.654,E2 -27152.654} C_VEL
LIN {X 0,Y 185.644,Z 394.634,A -85,B 0,C 180,E1 -27153.481,E2 -27153.481} C_VEL
LIN {X 0,Y 187.728,Z 388.725,A -85,B 0,C 180,E1 -27153.769,E2 -27153.769} C_VEL
LIN {X 0,Y 188.249,Z 386.909,A -85,B 0,C 180,E1 -27154.131,E2 -27154.131} C_VEL
LIN {X 0,Y 188.461,Z 385.584,A -85,B 0,C 180,E1 -27154.976,E2 -27154.976} C_VEL
LIN {X 0,Y 188.393,Z 384.62,A -85,B 0,C 180,E1 -27156.905,E2 -27156.905} C_VEL
LIN {X 0,Y 188.443,Z 384.221,A -85,B 0,C 180,E1 -27158.796,E2 -27158.796} C_VEL
LIN {X 0,Y 188.51,Z 384.478,A -85,B 0,C 180,E1 -27160.136,E2 -27160.136} C_VEL
LIN {X 0,Y 183.714,Z 397.853,A -85,B 0,C 180,E1 -27160.778,E2 -27160.778} C_VEL
LIN {X 0,Y 177.658,Z 410.432,A -85,B 0,C 180,E1 -27161.684,E2 -27161.684} C_VEL
LIN {X 0,Y 171.087,Z 421.283,A -85,B 0,C 180,E1 -27162.741,E2 -27162.741} C_VEL
LIN {X 0,Y 163.327,Z 431.822,A -85,B 0,C 180,E1 -27164.145,E2 -27164.145} C_VEL
LIN {X 0,Y 155.966,Z 440.171,A -85,B 0,C 180,E1 -27165.632,E2 -27165.632} C_VEL
LIN {X 0,Y 147.536,Z 448.239,A -85,B 0,C 180,E1 -27167.604,E2 -27167.604} C_VEL
LIN {X 0,Y 139.37,Z 454.853,A -85,B 0,C 180,E1 -27169.814,E2 -27169.814} C_VEL
LIN {X 0,Y 129.576,Z 461.476,A -85,B 0,C 180,E1 -27172.969,E2 -27172.969} C_VEL
LIN {X 0,Y 119.631,Z 466.936,A -85,B 0,C 180,E1 -27176.953,E2 -27176.953} C_VEL
LIN {X 0,Y 112.44,Z 470.093,A -85,B 0,C 180,E1 -27180.571,E2 -27180.571} C_VEL
LIN {X 0,Y 105.765,Z 472.375,A -85,B 0,C 180,E1 -27184.718,E2 -27184.718} C_VEL
LIN {X 0,Y 99.728,Z 473.863,A -85,B 0,C 180,E1 -27189.437,E2 -27189.437} C_VEL
LIN {X 0,Y 94.459,Z 474.569,A -85,B 0,C 180,E1 -27194.739,E2 -27194.739} C_VEL
LIN {X 0,Y 88.58,Z 474.171,A -85,B 0,C 180,E1 -27203.338,E2 -27203.338} C_VEL
LIN {X 0,Y 85.94,Z 473.059,A -85,B 0,C 180,E1 -27209.347,E2 -27209.347} C_VEL
LIN {X 0,Y 84.245,Z 471.266,A -85,B 0,C 180,E1 -27215.688,E2 -27215.688} C_VEL
LIN {X 0,Y 83.254,Z 467.341,A -85,B 0,C 180,E1 -27224.975,E2 -27224.975} C_VEL
LIN {X 0,Y 83.651,Z 463.473,A -85,B 0,C 180,E1 -27231.721,E2 -27231.721} C_VEL
LIN {X 0,Y 84.736,Z 458.558,A -85,B 0,C 180,E1 -27238.394,E2 -27238.394} C_VEL
LIN {X 0,Y 86.56,Z 452.373,A -85,B 0,C 180,E1 -27244.953,E2 -27244.953} C_VEL
LIN {X 0,Y 89.414,Z 444.117,A -85,B 0,C 180,E1 -27251.684,E2 -27251.684} C_VEL
LIN {X 0,Y 93.058,Z 434.504,A -85,B 0,C 180,E1 -27257.588,E2 -27257.588} C_VEL
LIN {X 0,Y 96.874,Z 423.981,A -85,B 0,C 180,E1 -27262.376,E2 -27262.376} C_VEL
LIN {X 0,Y 100.54,Z 413.35,A -85,B 0,C 180,E1 -27265.999,E2 -27265.999} C_VEL
LIN {X 0,Y 104.025,Z 401.446,A -85,B 0,C 180,E1 -27269.039,E2 -27269.039} C_VEL
LIN {X 0,Y 107.192,Z 388.332,A -85,B 0,C 180,E1 -27271.415,E2 -27271.415} C_VEL
LIN {X 0,Y 109.499,Z 375.285,A -85,B 0,C 180,E1 -27273.053,E2 -27273.053} C_VEL
LIN {X 0,Y 111.436,Z 359.155,A -85,B 0,C 180,E1 -27274.225,E2 -27274.225} C_VEL
LIN {X 0,Y 114.182,Z 328.594,A -85,B 0,C 180,E1 -27276.196,E2 -27276.196} C_VEL
LIN {X 0,Y 111.427,Z 319.725,A -85,B 0,C 180,E1 -27278.105,E2 -27278.105} C_VEL
LIN {X 0,Y 106.111,Z 307.22,A -85,B 0,C 180,E1 -27281.634,E2 -27281.634} C_VEL
LIN {X 0,Y 98.583,Z 294.035,A -85,B 0,C 180,E1 -27287.017,E2 -27287.017} C_VEL
LIN {X 0,Y 92.772,Z 285.601,A -85,B 0,C 180,E1 -27291.887,E2 -27291.887} C_VEL
LIN {X 0,Y 90.445,Z 282.461,A -85,B 0,C 180,E1 -27294.056,E2 -27294.056} C_VEL
LIN {X 0,Y 89.581,Z 281.148,A -85,B 0,C 180,E1 -27294.93,E2 -27294.93} C_VEL
LIN {X 0,Y 87.326,Z 278.696,A -85,B 0,C 180,E1 -27297.216,E2 -27297.216} C_VEL
LIN {X 0,Y 86.54,Z 276.723,A -85,B 0,C 180,E1 -27298.811,E2 -27298.811} C_VEL
LIN {X 0,Y 86.467,Z 276.201,A -85,B 0,C 180,E1 -27300.539,E2 -27300.539} C_VEL
LIN {X 0,Y 86.501,Z 276.208,A -85,B 0,C 180,E1 -27305.72,E2 -27305.72} C_VEL
LIN {X 0,Y 86.534,Z 276.205,A -85,B 0,C 180,E1 -27313.083,E2 -27313.083} C_VEL
LIN {X 0,Y 86.544,Z 276.195,A -85,B 0,C 180,E1 -27319.528,E2 -27319.528} C_VEL
LIN {X 0,Y 86.554,Z 276.179,A -85,B 0,C 180,E1 -27325.402,E2 -27325.402} C_VEL
LIN {X 0,Y 86.556,Z 276.18,A -85,B 0,C 180,E1 -27333.289,E2 -27333.289} C_VEL
LIN {X 0,Y 86.597,Z 276.185,A -85,B 0,C 180,E1 -27341.09,E2 -27341.09} C_VEL
LIN {X 0,Y 86.861,Z 276.147,A -85,B 0,C 180,E1 -27346.18,E2 -27346.18} C_VEL
LIN {X 0,Y 87.032,Z 276.128,A -85,B 0,C 180,E1 -27350.737,E2 -27350.737} C_VEL
LIN {X 0,Y 87.692,Z 276.029,A -85,B 0,C 180,E1 -27360.03,E2 -27360.03} C_VEL
LIN {X 0,Y 87.045,Z 276.091,A -85,B 0,C 180,E1 -27369.323,E2 -27369.323} C_VEL
LIN {X 0,Y 86.763,Z 276.277,A -85,B 0,C 180,E1 -27376.5,E2 -27376.5} C_VEL
LIN {X 0,Y 87.014,Z 277.482,A -85,B 0,C 180,E1 -27377.965,E2 -27377.965} C_VEL
LIN {X 0,Y 88.706,Z 280.262,A -85,B 0,C 180,E1 -27380.009,E2 -27380.009} C_VEL
LIN {X 0,Y 90.082,Z 281.603,A -85,B 0,C 180,E1 -27381.331,E2 -27381.331} C_VEL
LIN {X 0,Y 92.166,Z 284.956,A -85,B 0,C 180,E1 -27383.388,E2 -27383.388} C_VEL
LIN {X 0,Y 93.648,Z 286.974,A -85,B 0,C 180,E1 -27384.707,E2 -27384.707} C_VEL
LIN {X 0,Y 96.231,Z 290.968,A -85,B 0,C 180,E1 -27386.93,E2 -27386.93} C_VEL
LIN {X 0,Y 101.075,Z 299.117,A -85,B 0,C 180,E1 -27390.77,E2 -27390.77} C_VEL
LIN {X 0,Y 107.753,Z 312.221,A -85,B 0,C 180,E1 -27395.397,E2 -27395.397} C_VEL
LIN {X 0,Y 111.566,Z 323.412,A -85,B 0,C 180,E1 -27398.1,E2 -27398.1} C_VEL
LIN {X 0,Y 114.162,Z 332.108,A -85,B 0,C 180,E1 -27399.909,E2 -27399.909} C_VEL
LIN {X 0,Y 110.083,Z 373.587,A -85,B 0,C 180,E1 -27402.584,E2 -27402.584} C_VEL
LIN {X 0,Y 107.894,Z 387.132,A -85,B 0,C 180,E1 -27404.057,E2 -27404.057} C_VEL
LIN {X 0,Y 105.161,Z 399.671,A -85,B 0,C 180,E1 -27406.094,E2 -27406.094} C_VEL
LIN {X 0,Y 101.572,Z 412.03,A -85,B 0,C 180,E1 -27408.896,E2 -27408.896} C_VEL
LIN {X 0,Y 97.78,Z 423.7,A -85,B 0,C 180,E1 -27412.557,E2 -27412.557} C_VEL
LIN {X 0,Y 93.84,Z 434.411,A -85,B 0,C 180,E1 -27417.105,E2 -27417.105} C_VEL
LIN {X 0,Y 90.426,Z 443.442,A -85,B 0,C 180,E1 -27422.196,E2 -27422.196} C_VEL
LIN {X 0,Y 87.25,Z 452.231,A -85,B 0,C 180,E1 -27428.74,E2 -27428.74} C_VEL
LIN {X 0,Y 85.214,Z 459.225,A -85,B 0,C 180,E1 -27435.667,E2 -27435.667} C_VEL
LIN {X 0,Y 84.187,Z 464.783,A -85,B 0,C 180,E1 -27442.798,E2 -27442.798} C_VEL
LIN {X 0,Y 84.019,Z 469.092,A -85,B 0,C 180,E1 -27449.992,E2 -27449.992} C_VEL
LIN {X 0,Y 84.015,Z 471.308,A -85,B 0,C 180,E1 -27454.79,E2 -27454.79} C_VEL
LIN {X 0,Y 85.222,Z 474.487,A -85,B 0,C 180,E1 -27464.315,E2 -27464.315} C_VEL
LIN {X 0,Y 88.484,Z 476.077,A -85,B 0,C 180,E1 -27473.39,E2 -27473.39} C_VEL
LIN {X 0,Y 93.853,Z 476.255,A -85,B 0,C 180,E1 -27481.604,E2 -27481.604} C_VEL
LIN {X 0,Y 101.138,Z 474.99,A -85,B 0,C 180,E1 -27488.702,E2 -27488.702} C_VEL
LIN {X 0,Y 109.858,Z 472.221,A -85,B 0,C 180,E1 -27494.715,E2 -27494.715} C_VEL
LIN {X 0,Y 117.036,Z 469.151,A -85,B 0,C 180,E1 -27498.632,E2 -27498.632} C_VEL
LIN {X 0,Y 127.416,Z 463.568,A -85,B 0,C 180,E1 -27503.1,E2 -27503.1} C_VEL
LIN {X 0,Y 137.216,Z 457.066,A -85,B 0,C 180,E1 -27506.325,E2 -27506.325} C_VEL
LIN {X 0,Y 146.012,Z 450.092,A -85,B 0,C 180,E1 -27508.679,E2 -27508.679} C_VEL
LIN {X 0,Y 155.035,Z 441.551,A -85,B 0,C 180,E1 -27510.756,E2 -27510.756} C_VEL
LIN {X 0,Y 162.727,Z 432.889,A -85,B 0,C 180,E1 -27512.286,E2 -27512.286} C_VEL
LIN {X 0,Y 170.604,Z 422.287,A -85,B 0,C 180,E1 -27513.625,E2 -27513.625} C_VEL
LIN {X 0,Y 176.966,Z 411.902,A -85,B 0,C 180,E1 -27514.61,E2 -27514.61} C_VEL
LIN {X 0,Y 182.787,Z 400.166,A -85,B 0,C 180,E1 -27515.38,E2 -27515.38} C_VEL
LIN {X 0,Y 187.297,Z 388.49,A -85,B 0,C 180,E1 -27515.954,E2 -27515.954} C_VEL
LIN {X 0,Y 188.379,Z 385.01,A -85,B 0,C 180,E1 -27516.138,E2 -27516.138} C_VEL
LIN {X 0,Y 188.393,Z 384.62,A -85,B 0,C 180,E1 -27516.905,E2 -27516.905} C_VEL
LIN {X 0,Y 188.199,Z 385.052,A -85,B 0,C 180,E1 -27517.645,E2 -27517.645} C_VEL
LIN {X 0,Y 187.51,Z 387.166,A -85,B 0,C 180,E1 -27518.455,E2 -27518.455} C_VEL
LIN {X 0,Y 186.167,Z 391.138,A -85,B 0,C 180,E1 -27519.145,E2 -27519.145} C_VEL
LIN {X 0,Y 184.824,Z 394.68,A -85,B 0,C 180,E1 -27519.403,E2 -27519.403} C_VEL
LIN {X 0,Y 180.674,Z 404.064,A -85,B 0,C 180,E1 -27519.364,E2 -27519.364} C_VEL
LIN {X 0,Y 177.206,Z 410.644,A -85,B 0,C 180,E1 -27519.409,E2 -27519.409} C_VEL
LIN {X 0,Y 176.02,Z 412.743,A -85,B 0,C 180,E1 -27519.542,E2 -27519.542} C_VEL
LIN {X 0,Y 169.032,Z 423.586,A -85,B 0,C 180,E1 -27520.557,E2 -27520.557} C_VEL
LIN {X 0,Y 160.149,Z 434.734,A -85,B 0,C 180,E1 -27522.024,E2 -27522.024} C_VEL
LIN {X 0,Y 153.001,Z 442.192,A -85,B 0,C 180,E1 -27523.336,E2 -27523.336} C_VEL
LIN {X 0,Y 143.546,Z 450.591,A -85,B 0,C 180,E1 -27525.387,E2 -27525.387} C_VEL
LIN {X 0,Y 133.871,Z 457.663,A -85,B 0,C 180,E1 -27527.859,E2 -27527.859} C_VEL
LIN {X 0,Y 123.18,Z 464.012,A -85,B 0,C 180,E1 -27531.221,E2 -27531.221} C_VEL
LIN {X 0,Y 112.807,Z 468.856,A -85,B 0,C 180,E1 -27535.338,E2 -27535.338} C_VEL
LIN {X 0,Y 103.882,Z 471.998,A -85,B 0,C 180,E1 -27539.975,E2 -27539.975} C_VEL
LIN {X 0,Y 97.613,Z 473.6,A -85,B 0,C 180,E1 -27544.101,E2 -27544.101} C_VEL
LIN {X 0,Y 91.993,Z 474.48,A -85,B 0,C 180,E1 -27548.759,E2 -27548.759} C_VEL
LIN {X 0,Y 86.954,Z 474.737,A -85,B 0,C 180,E1 -27554.131,E2 -27554.131} C_VEL
LIN {X 0,Y 82.56,Z 474.216,A -85,B 0,C 180,E1 -27560.574,E2 -27560.574} C_VEL
LIN {X 0,Y 79.267,Z 472.879,A -85,B 0,C 180,E1 -27567.568,E2 -27567.568} C_VEL
LIN {X 0,Y 77.222,Z 470.74,A -85,B 0,C 180,E1 -27575.023,E2 -27575.023} C_VEL
LIN {X 0,Y 76.2,Z 466.774,A -85,B 0,C 180,E1 -27584.781,E2 -27584.781} C_VEL
LIN {X 0,Y 76.701,Z 462.314,A -85,B 0,C 180,E1 -27592.793,E2 -27592.793} C_VEL
LIN {X 0,Y 78.024,Z 456.89,A -85,B 0,C 180,E1 -27600.285,E2 -27600.285} C_VEL
LIN {X 0,Y 80.489,Z 449.36,A -85,B 0,C 180,E1 -27608.226,E2 -27608.226} C_VEL
LIN {X 0,Y 83.974,Z 440.096,A -85,B 0,C 180,E1 -27615.467,E2 -27615.467} C_VEL
LIN {X 0,Y 87.555,Z 431.047,A -85,B 0,C 180,E1 -27620.77,E2 -27620.77} C_VEL
LIN {X 0,Y 91.885,Z 419.801,A -85,B 0,C 180,E1 -27625.621,E2 -27625.621} C_VEL
LIN {X 0,Y 96.037,Z 407.559,A -85,B 0,C 180,E1 -27629.483,E2 -27629.483} C_VEL
LIN {X 0,Y 99.392,Z 395.545,A -85,B 0,C 180,E1 -27632.21,E2 -27632.21} C_VEL
LIN {X 0,Y 102.267,Z 382.593,A -85,B 0,C 180,E1 -27634.29,E2 -27634.29} C_VEL
LIN {X 0,Y 104.489,Z 369.177,A -85,B 0,C 180,E1 -27635.656,E2 -27635.656} C_VEL
LIN {X 0,Y 108.364,Z 330.238,A -85,B 0,C 180,E1 -27638.252,E2 -27638.252} C_VEL
LIN {X 0,Y 106.18,Z 323.129,A -85,B 0,C 180,E1 -27639.878,E2 -27639.878} C_VEL
LIN {X 0,Y 101.313,Z 311.333,A -85,B 0,C 180,E1 -27643.443,E2 -27643.443} C_VEL
LIN {X 0,Y 94.659,Z 299.236,A -85,B 0,C 180,E1 -27648.715,E2 -27648.715} C_VEL
LIN {X 0,Y 89.124,Z 290.993,A -85,B 0,C 180,E1 -27653.754,E2 -27653.754} C_VEL
LIN {X 0,Y 86.092,Z 286.756,A -85,B 0,C 180,E1 -27656.934,E2 -27656.934} C_VEL
LIN {X 0,Y 83.713,Z 283.538,A -85,B 0,C 180,E1 -27659.761,E2 -27659.761} C_VEL
LIN {X 0,Y 83.233,Z 282.523,A -85,B 0,C 180,E1 -27660.448,E2 -27660.448} C_VEL
LIN {X 0,Y 80.66,Z 280.232,A -85,B 0,C 180,E1 -27663.831,E2 -27663.831} C_VEL
LIN {X 0,Y 79.572,Z 277.826,A -85,B 0,C 180,E1 -27666.065,E2 -27666.065} C_VEL
LIN {X 0,Y 79.404,Z 277.13,A -85,B 0,C 180,E1 -27668.295,E2 -27668.295} C_VEL
LIN {X 0,Y 79.444,Z 277.07,A -85,B 0,C 180,E1 -27675.061,E2 -27675.061} C_VEL
LIN {X 0,Y 79.442,Z 277.074,A -85,B 0,C 180,E1 -27682.783,E2 -27682.783} C_VEL
LIN {X 0,Y 79.458,Z 277.069,A -85,B 0,C 180,E1 -27692.206,E2 -27692.206} C_VEL
LIN {X 0,Y 79.473,Z 277.085,A -85,B 0,C 180,E1 -27699.321,E2 -27699.321} C_VEL
LIN {X 0,Y 79.784,Z 277.024,A -85,B 0,C 180,E1 -27705.719,E2 -27705.719} C_VEL
LIN {X 0,Y 79.915,Z 277.019,A -85,B 0,C 180,E1 -27709.904,E2 -27709.904} C_VEL
LIN {X 0,Y 80.622,Z 276.904,A -85,B 0,C 180,E1 -27720.033,E2 -27720.033} C_VEL
LIN {X 0,Y 80.04,Z 277.191,A -85,B 0,C 180,E1 -27729.19,E2 -27729.19} C_VEL
LIN {X 0,Y 80.274,Z 278.547,A -85,B 0,C 180,E1 -27731.06,E2 -27731.06} C_VEL
LIN {X 0,Y 81.655,Z 280.951,A -85,B 0,C 180,E1 -27733.251,E2 -27733.251} C_VEL
LIN {X 0,Y 83.603,Z 282.779,A -85,B 0,C 180,E1 -27735.731,E2 -27735.731} C_VEL
LIN {X 0,Y 85.594,Z 286.082,A -85,B 0,C 180,E1 -27738.274,E2 -27738.274} C_VEL
LIN {X 0,Y 86.986,Z 287.831,A -85,B 0,C 180,E1 -27739.806,E2 -27739.806} C_VEL
LIN {X 0,Y 90.486,Z 293.202,A -85,B 0,C 180,E1 -27743.401,E2 -27743.401} C_VEL
LIN {X 0,Y 94.834,Z 300.261,A -85,B 0,C 180,E1 -27747.309,E2 -27747.309} C_VEL
LIN {X 0,Y 100.131,Z 310.532,A -85,B 0,C 180,E1 -27751.644,E2 -27751.644} C_VEL
LIN {X 0,Y 103.635,Z 318.316,A -85,B 0,C 180,E1 -27754.249,E2 -27754.249} C_VEL
LIN {X 0,Y 108.277,Z 333.632,A -85,B 0,C 180,E1 -27757.846,E2 -27757.846} C_VEL
LIN {X 0,Y 104.139,Z 373.783,A -85,B 0,C 180,E1 -27760.521,E2 -27760.521} C_VEL
LIN {X 0,Y 101.801,Z 387.476,A -85,B 0,C 180,E1 -27762.077,E2 -27762.077} C_VEL
LIN {X 0,Y 99.067,Z 399.329,A -85,B 0,C 180,E1 -27764.078,E2 -27764.078} C_VEL
LIN {X 0,Y 95.306,Z 411.707,A -85,B 0,C 180,E1 -27766.983,E2 -27766.983} C_VEL
LIN {X 0,Y 91.205,Z 423.626,A -85,B 0,C 180,E1 -27770.904,E2 -27770.904} C_VEL
LIN {X 0,Y 87.155,Z 434.108,A -85,B 0,C 180,E1 -27775.626,E2 -27775.626} C_VEL
LIN {X 0,Y 83.545,Z 443.139,A -85,B 0,C 180,E1 -27781.063,E2 -27781.063} C_VEL
LIN {X 0,Y 80.217,Z 451.965,A -85,B 0,C 180,E1 -27788.13,E2 -27788.13} C_VEL
LIN {X 0,Y 78.096,Z 458.992,A -85,B 0,C 180,E1 -27795.663,E2 -27795.663} C_VEL
LIN {X 0,Y 77.014,Z 465.373,A -85,B 0,C 180,E1 -27804.755,E2 -27804.755} C_VEL
LIN {X 0,Y 76.974,Z 468.279,A -85,B 0,C 180,E1 -27809.991,E2 -27809.991} C_VEL
LIN {X 0,Y 76.991,Z 470.605,A -85,B 0,C 180,E1 -27815.228,E2 -27815.228} C_VEL
LIN {X 0,Y 78.372,Z 473.962,A -85,B 0,C 180,E1 -27825.597,E2 -27825.597} C_VEL
LIN {X 0,Y 81.989,Z 475.824,A -85,B 0,C 180,E1 -27835.369,E2 -27835.369} C_VEL
LIN {X 0,Y 87.879,Z 476.204,A -85,B 0,C 180,E1 -27844.033,E2 -27844.033} C_VEL
LIN {X 0,Y 95.696,Z 475.182,A -85,B 0,C 180,E1 -27851.363,E2 -27851.363} C_VEL
LIN {X 0,Y 104.949,Z 472.708,A -85,B 0,C 180,E1 -27857.434,E2 -27857.434} C_VEL
LIN {X 0,Y 115.147,Z 468.655,A -85,B 0,C 180,E1 -27862.499,E2 -27862.499} C_VEL
LIN {X 0,Y 123.333,Z 464.566,A -85,B 0,C 180,E1 -27865.706,E2 -27865.706} C_VEL
LIN {X 0,Y 131.998,Z 459.393,A -85,B 0,C 180,E1 -27868.406,E2 -27868.406} C_VEL
LIN {X 0,Y 140.999,Z 452.98,A -85,B 0,C 180,E1 -27870.713,E2 -27870.713} C_VEL
LIN {X 0,Y 150.231,Z 445.122,A -85,B 0,C 180,E1 -27872.717,E2 -27872.717} C_VEL
LIN {X 0,Y 158.069,Z 437.259,A -85,B 0,C 180,E1 -27874.192,E2 -27874.192} C_VEL
LIN {X 0,Y 166.073,Z 427.756,A -85,B 0,C 180,E1 -27875.473,E2 -27875.473} C_VEL
LIN {X 0,Y 174.158,Z 415.929,A -85,B 0,C 180,E1 -27876.632,E2 -27876.632} C_VEL
LIN {X 0,Y 180.737,Z 403.924,A -85,B 0,C 180,E1 -27877.435,E2 -27877.435} C_VEL
LIN {X 0,Y 184.868,Z 394.426,A -85,B 0,C 180,E1 -27877.904,E2 -27877.904} C_VEL
LIN {X 0,Y 184.958,Z 394.176,A -85,B 0,C 180,E1 -27878.377,E2 -27878.377} C_VEL
LIN {X 0,Y 179.673,Z 405.969,A -85,B 0,C 180,E1 -27879.036,E2 -27879.036} C_VEL
LIN {X 0,Y 176.02,Z 412.743,A -85,B 0,C 180,E1 -27879.542,E2 -27879.542} C_VEL
LIN {X 0,Y 172.99,Z 417.778,A -85,B 0,C 180,E1 -27879.766,E2 -27879.766} C_VEL
LIN {X 0,Y 167.268,Z 425.873,A -85,B 0,C 180,E1 -27879.598,E2 -27879.598} C_VEL
LIN {X 0,Y 160.959,Z 433.483,A -85,B 0,C 180,E1 -27879.486,E2 -27879.486} C_VEL
LIN {X 0,Y 157.011,Z 437.734,A -85,B 0,C 180,E1 -27879.834,E2 -27879.834} C_VEL
LIN {X 0,Y 148.368,Z 445.964,A -85,B 0,C 180,E1 -27881.312,E2 -27881.312} C_VEL
LIN {X 0,Y 139.558,Z 452.997,A -85,B 0,C 180,E1 -27883.081,E2 -27883.081} C_VEL
LIN {X 0,Y 130.875,Z 458.815,A -85,B 0,C 180,E1 -27885.127,E2 -27885.127} C_VEL
LIN {X 0,Y 122.368,Z 463.629,A -85,B 0,C 180,E1 -27887.489,E2 -27887.489} C_VEL
LIN {X 0,Y 111.422,Z 468.616,A -85,B 0,C 180,E1 -27891.266,E2 -27891.266} C_VEL
LIN {X 0,Y 101.058,Z 472.072,A -85,B 0,C 180,E1 -27895.986,E2 -27895.986} C_VEL
LIN {X 0,Y 91.402,Z 474.157,A -85,B 0,C 180,E1 -27901.916,E2 -27901.916} C_VEL
LIN {X 0,Y 82.517,Z 474.861,A -85,B 0,C 180,E1 -27909.774,E2 -27909.774} C_VEL
LIN {X 0,Y 77.831,Z 474.437,A -85,B 0,C 180,E1 -27915.681,E2 -27915.681} C_VEL
LIN {X 0,Y 74.088,Z 473.394,A -85,B 0,C 180,E1 -27922.259,E2 -27922.259} C_VEL
LIN {X 0,Y 70.495,Z 470.614,A -85,B 0,C 180,E1 -27932.878,E2 -27932.878} C_VEL
LIN {X 0,Y 69.32,Z 467.707,A -85,B 0,C 180,E1 -27940.872,E2 -27940.872} C_VEL
LIN {X 0,Y 69.403,Z 462.894,A -85,B 0,C 180,E1 -27950.886,E2 -27950.886} C_VEL
LIN {X 0,Y 70.836,Z 456.851,A -85,B 0,C 180,E1 -27960.271,E2 -27960.271} C_VEL
LIN {X 0,Y 73.189,Z 449.94,A -85,B 0,C 180,E1 -27968.356,E2 -27968.356} C_VEL
LIN {X 0,Y 76.285,Z 442.083,A -85,B 0,C 180,E1 -27975.29,E2 -27975.29} C_VEL
LIN {X 0,Y 80.458,Z 432.086,A -85,B 0,C 180,E1 -27981.848,E2 -27981.848} C_VEL
LIN {X 0,Y 84.79,Z 421.467,A -85,B 0,C 180,E1 -27986.923,E2 -27986.923} C_VEL
LIN {X 0,Y 88.935,Z 410.159,A -85,B 0,C 180,E1 -27990.836,E2 -27990.836} C_VEL
LIN {X 0,Y 92.875,Z 397.443,A -85,B 0,C 180,E1 -27994.027,E2 -27994.027} C_VEL
LIN {X 0,Y 96.023,Z 384.265,A -85,B 0,C 180,E1 -27996.31,E2 -27996.31} C_VEL
LIN {X 0,Y 98.469,Z 370.449,A -85,B 0,C 180,E1 -27997.859,E2 -27997.859} C_VEL
LIN {X 0,Y 102.597,Z 331.746,A -85,B 0,C 180,E1 -28000.486,E2 -28000.486} C_VEL
LIN {X 0,Y 100.903,Z 326.245,A -85,B 0,C 180,E1 -28001.895,E2 -28001.895} C_VEL
LIN {X 0,Y 96.682,Z 315.559,A -85,B 0,C 180,E1 -28005.383,E2 -28005.383} C_VEL
LIN {X 0,Y 90.643,Z 304.246,A -85,B 0,C 180,E1 -28010.623,E2 -28010.623} C_VEL
LIN {X 0,Y 85.686,Z 296.577,A -85,B 0,C 180,E1 -28015.628,E2 -28015.628} C_VEL
LIN {X 0,Y 82.852,Z 292.411,A -85,B 0,C 180,E1 -28018.96,E2 -28018.96} C_VEL
LIN {X 0,Y 80.102,Z 288.463,A -85,B 0,C 180,E1 -28022.701,E2 -28022.701} C_VEL
LIN {X 0,Y 77.67,Z 285.671,A -85,B 0,C 180,E1 -28026.371,E2 -28026.371} C_VEL
LIN {X 0,Y 76.749,Z 283.747,A -85,B 0,C 180,E1 -28028.146,E2 -28028.146} C_VEL
LIN {X 0,Y 74.008,Z 281.791,A -85,B 0,C 180,E1 -28033.244,E2 -28033.244} C_VEL
LIN {X 0,Y 72.397,Z 278.644,A -85,B 0,C 180,E1 -28038.337,E2 -28038.337} C_VEL
LIN {X 0,Y 72.337,Z 278.01,A -85,B 0,C 180,E1 -28041.024,E2 -28041.024} C_VEL
LIN {X 0,Y 72.325,Z 277.965,A -85,B 0,C 180,E1 -28044.384,E2 -28044.384} C_VEL
LIN {X 0,Y 72.361,Z 277.962,A -85,B 0,C 180,E1 -28050.991,E2 -28050.991} C_VEL
LIN {X 0,Y 72.361,Z 277.953,A -85,B 0,C 180,E1 -28057.18,E2 -28057.18} C_VEL
LIN {X 0,Y 72.677,Z 277.907,A -85,B 0,C 180,E1 -28065.279,E2 -28065.279} C_VEL
LIN {X 0,Y 72.813,Z 277.912,A -85,B 0,C 180,E1 -28068.907,E2 -28068.907} C_VEL
LIN {X 0,Y 73.411,Z 278.172,A -85,B 0,C 180,E1 -28078.665,E2 -28078.665} C_VEL
LIN {X 0,Y 73.65,Z 278.441,A -85,B 0,C 180,E1 -28080.036,E2 -28080.036} C_VEL
LIN {X 0,Y 74.578,Z 281.227,A -85,B 0,C 180,E1 -28083.412,E2 -28083.412} C_VEL
LIN {X 0,Y 76.805,Z 283.329,A -85,B 0,C 180,E1 -28087.593,E2 -28087.593} C_VEL
LIN {X 0,Y 77.399,Z 284.232,A -85,B 0,C 180,E1 -28088.684,E2 -28088.684} C_VEL
LIN {X 0,Y 79.097,Z 287.128,A -85,B 0,C 180,E1 -28091.591,E2 -28091.591} C_VEL
LIN {X 0,Y 80.847,Z 289.093,A -85,B 0,C 180,E1 -28094.046,E2 -28094.046} C_VEL
LIN {X 0,Y 83.204,Z 292.641,A -85,B 0,C 180,E1 -28097.188,E2 -28097.188} C_VEL
LIN {X 0,Y 87.046,Z 298.799,A -85,B 0,C 180,E1 -28101.646,E2 -28101.646} C_VEL
LIN {X 0,Y 91.819,Z 307.138,A -85,B 0,C 180,E1 -28106.36,E2 -28106.36} C_VEL
LIN {X 0,Y 96.681,Z 317.26,A -85,B 0,C 180,E1 -28110.617,E2 -28110.617} C_VEL
LIN {X 0,Y 98.822,Z 322.488,A -85,B 0,C 180,E1 -28112.407,E2 -28112.407} C_VEL
LIN {X 0,Y 102.433,Z 334.987,A -85,B 0,C 180,E1 -28115.572,E2 -28115.572} C_VEL
LIN {X 0,Y 98.811,Z 369.82,A -85,B 0,C 180,E1 -28117.944,E2 -28117.944} C_VEL
LIN {X 0,Y 96.589,Z 383.863,A -85,B 0,C 180,E1 -28119.357,E2 -28119.357} C_VEL
LIN {X 0,Y 93.694,Z 396.547,A -85,B 0,C 180,E1 -28121.391,E2 -28121.391} C_VEL
LIN {X 0,Y 90.239,Z 407.936,A -85,B 0,C 180,E1 -28123.902,E2 -28123.902} C_VEL
LIN {X 0,Y 86.129,Z 419.777,A -85,B 0,C 180,E1 -28127.577,E2 -28127.577} C_VEL
LIN {X 0,Y 81.831,Z 430.634,A -85,B 0,C 180,E1 -28132.261,E2 -28132.261} C_VEL
LIN {X 0,Y 77.403,Z 441.188,A -85,B 0,C 180,E1 -28138.518,E2 -28138.518} C_VEL
LIN {X 0,Y 73.683,Z 450.328,A -85,B 0,C 180,E1 -28146.076,E2 -28146.076} C_VEL
LIN {X 0,Y 71.249,Z 457.682,A -85,B 0,C 180,E1 -28154.251,E2 -28154.251} C_VEL
LIN {X 0,Y 70.142,Z 462.606,A -85,B 0,C 180,E1 -28161.346,E2 -28161.346} C_VEL
LIN {X 0,Y 69.936,Z 467.339,A -85,B 0,C 180,E1 -28169.99,E2 -28169.99} C_VEL
LIN {X 0,Y 70.1,Z 470.849,A -85,B 0,C 180,E1 -28178.639,E2 -28178.639} C_VEL
LIN {X 0,Y 71.575,Z 473.415,A -85,B 0,C 180,E1 -28187.122,E2 -28187.122} C_VEL
LIN {X 0,Y 75.613,Z 475.485,A -85,B 0,C 180,E1 -28197.682,E2 -28197.682} C_VEL
LIN {X 0,Y 82.089,Z 476.146,A -85,B 0,C 180,E1 -28206.809,E2 -28206.809} C_VEL
LIN {X 0,Y 90.488,Z 475.347,A -85,B 0,C 180,E1 -28214.336,E2 -28214.336} C_VEL
LIN {X 0,Y 100.301,Z 473.118,A -85,B 0,C 180,E1 -28220.41,E2 -28220.41} C_VEL
LIN {X 0,Y 107.278,Z 470.839,A -85,B 0,C 180,E1 -28223.843,E2 -28223.843} C_VEL
LIN {X 0,Y 116.606,Z 466.952,A -85,B 0,C 180,E1 -28227.531,E2 -28227.531} C_VEL
LIN {X 0,Y 125.441,Z 462.41,A -85,B 0,C 180,E1 -28230.262,E2 -28230.262} C_VEL
LIN {X 0,Y 136.159,Z 455.683,A -85,B 0,C 180,E1 -28232.908,E2 -28232.908} C_VEL
LIN {X 0,Y 145.601,Z 448.51,A -85,B 0,C 180,E1 -28234.816,E2 -28234.816} C_VEL
LIN {X 0,Y 155.21,Z 439.705,A -85,B 0,C 180,E1 -28236.469,E2 -28236.469} C_VEL
LIN {X 0,Y 163.938,Z 429.966,A -85,B 0,C 180,E1 -28237.742,E2 -28237.742} C_VEL
LIN {X 0,Y 166.635,Z 426.566,A -85,B 0,C 180,E1 -28238.092,E2 -28238.092} C_VEL
LIN {X 0,Y 166.196,Z 427.141,A -85,B 0,C 180,E1 -28238.472,E2 -28238.472} C_VEL
LIN {X 0,Y 158.875,Z 435.788,A -85,B 0,C 180,E1 -28239.537,E2 -28239.537} C_VEL
LIN {X 0,Y 157.011,Z 437.734,A -85,B 0,C 180,E1 -28239.834,E2 -28239.834} C_VEL
LIN {X 0,Y 152.857,Z 441.87,A -85,B 0,C 180,E1 -28240.24,E2 -28240.24} C_VEL
LIN {X 0,Y 145.342,Z 448.378,A -85,B 0,C 180,E1 -28240.363,E2 -28240.363} C_VEL
LIN {X 0,Y 137.452,Z 454.24,A -85,B 0,C 180,E1 -28240.614,E2 -28240.614} C_VEL
LIN {X 0,Y 132.743,Z 457.308,A -85,B 0,C 180,E1 -28241.28,E2 -28241.28} C_VEL
LIN {X 0,Y 123.35,Z 462.677,A -85,B 0,C 180,E1 -28243.427,E2 -28243.427} C_VEL
LIN {X 0,Y 111.217,Z 468.116,A -85,B 0,C 180,E1 -28246.935,E2 -28246.935} C_VEL
LIN {X 0,Y 99.484,Z 471.995,A -85,B 0,C 180,E1 -28251.45,E2 -28251.45} C_VEL
LIN {X 0,Y 91.404,Z 473.787,A -85,B 0,C 180,E1 -28255.561,E2 -28255.561} C_VEL
LIN {X 0,Y 84.323,Z 474.716,A -85,B 0,C 180,E1 -28260.176,E2 -28260.176} C_VEL
LIN {X 0,Y 77.7,Z 474.947,A -85,B 0,C 180,E1 -28265.851,E2 -28265.851} C_VEL
LIN {X 0,Y 71.981,Z 474.402,A -85,B 0,C 180,E1 -28272.528,E2 -28272.528} C_VEL
LIN {X 0,Y 67.434,Z 473.024,A -85,B 0,C 180,E1 -28280.315,E2 -28280.315} C_VEL
LIN {X 0,Y 64.236,Z 470.857,A -85,B 0,C 180,E1 -28288.946,E2 -28288.946} C_VEL
LIN {X 0,Y 62.495,Z 467.877,A -85,B 0,C 180,E1 -28298.095,E2 -28298.095} C_VEL
LIN {X 0,Y 62.273,Z 462.773,A -85,B 0,C 180,E1 -28309.885,E2 -28309.885} C_VEL
LIN {X 0,Y 63.431,Z 457.506,A -85,B 0,C 180,E1 -28319.066,E2 -28319.066} C_VEL
LIN {X 0,Y 65.706,Z 450.884,A -85,B 0,C 180,E1 -28327.927,E2 -28327.927} C_VEL
LIN {X 0,Y 68.602,Z 443.786,A -85,B 0,C 180,E1 -28335.171,E2 -28335.171} C_VEL
LIN {X 0,Y 72.877,Z 434.256,A -85,B 0,C 180,E1 -28342.39,E2 -28342.39} C_VEL
LIN {X 0,Y 77.627,Z 423.23,A -85,B 0,C 180,E1 -28348.362,E2 -28348.362} C_VEL
LIN {X 0,Y 81.94,Z 412.594,A -85,B 0,C 180,E1 -28352.469,E2 -28352.469} C_VEL
LIN {X 0,Y 86.043,Z 400.362,A -85,B 0,C 180,E1 -28355.868,E2 -28355.868} C_VEL
LIN {X 0,Y 89.331,Z 388.442,A -85,B 0,C 180,E1 -28358.206,E2 -28358.206} C_VEL
LIN {X 0,Y 91.956,Z 375.568,A -85,B 0,C 180,E1 -28359.957,E2 -28359.957} C_VEL
LIN {X 0,Y 94.22,Z 359.218,A -85,B 0,C 180,E1 -28361.207,E2 -28361.207} C_VEL
LIN {X 0,Y 96.967,Z 333.846,A -85,B 0,C 180,E1 -28362.936,E2 -28362.936} C_VEL
LIN {X 0,Y 96.046,Z 330.164,A -85,B 0,C 180,E1 -28363.878,E2 -28363.878} C_VEL
LIN {X 0,Y 92.133,Z 319.86,A -85,B 0,C 180,E1 -28367.446,E2 -28367.446} C_VEL
LIN {X 0,Y 86.828,Z 309.409,A -85,B 0,C 180,E1 -28372.61,E2 -28372.61} C_VEL
LIN {X 0,Y 82.198,Z 301.867,A -85,B 0,C 180,E1 -28377.851,E2 -28377.851} C_VEL
LIN {X 0,Y 79.663,Z 298.014,A -85,B 0,C 180,E1 -28381.181,E2 -28381.181} C_VEL
LIN {X 0,Y 77.274,Z 294.428,A -85,B 0,C 180,E1 -28384.819,E2 -28384.819} C_VEL
LIN {X 0,Y 74.942,Z 291.318,A -85,B 0,C 180,E1 -28388.876,E2 -28388.876} C_VEL
LIN {X 0,Y 74.334,Z 290.193,A -85,B 0,C 180,E1 -28390.166,E2 -28390.166} C_VEL
LIN {X 0,Y 71.993,Z 288.179,A -85,B 0,C 180,E1 -28395.064,E2 -28395.064} C_VEL
LIN {X 0,Y 70.276,Z 284.927,A -85,B 0,C 180,E1 -28400.651,E2 -28400.651} C_VEL
LIN {X 0,Y 67.873,Z 283.525,A -85,B 0,C 180,E1 -28412.536,E2 -28412.536} C_VEL
LIN {X 0,Y 68.257,Z 283.431,A -85,B 0,C 180,E1 -28426.123,E2 -28426.123} C_VEL
LIN {X 0,Y 71.462,Z 284.971,A -85,B 0,C 180,E1 -28438.274,E2 -28438.274} C_VEL
LIN {X 0,Y 72.807,Z 288.058,A -85,B 0,C 180,E1 -28442.284,E2 -28442.284} C_VEL
LIN {X 0,Y 74.844,Z 290.229,A -85,B 0,C 180,E1 -28446.437,E2 -28446.437} C_VEL
LIN {X 0,Y 76.859,Z 293.632,A -85,B 0,C 180,E1 -28450.239,E2 -28450.239} C_VEL
LIN {X 0,Y 78.027,Z 295.15,A -85,B 0,C 180,E1 -28452.081,E2 -28452.081} C_VEL
LIN {X 0,Y 80.771,Z 299.571,A -85,B 0,C 180,E1 -28456.074,E2 -28456.074} C_VEL
LIN {X 0,Y 84.414,Z 305.585,A -85,B 0,C 180,E1 -28460.585,E2 -28460.585} C_VEL
LIN {X 0,Y 88.597,Z 313.737,A -85,B 0,C 180,E1 -28465.142,E2 -28465.142} C_VEL
LIN {X 0,Y 93.581,Z 324.879,A -85,B 0,C 180,E1 -28469.84,E2 -28469.84} C_VEL
LIN {X 0,Y 96.781,Z 336.495,A -85,B 0,C 180,E1 -28473.069,E2 -28473.069} C_VEL
LIN {X 0,Y 93.186,Z 369.624,A -85,B 0,C 180,E1 -28475.383,E2 -28475.383} C_VEL
LIN {X 0,Y 90.995,Z 383.004,A -85,B 0,C 180,E1 -28476.733,E2 -28476.733} C_VEL
LIN {X 0,Y 87.926,Z 395.899,A -85,B 0,C 180,E1 -28478.789,E2 -28478.789} C_VEL
LIN {X 0,Y 84.307,Z 407.41,A -85,B 0,C 180,E1 -28481.376,E2 -28481.376} C_VEL
LIN {X 0,Y 79.879,Z 419.51,A -85,B 0,C 180,E1 -28485.251,E2 -28485.251} C_VEL
LIN {X 0,Y 75.387,Z 430.253,A -85,B 0,C 180,E1 -28490.128,E2 -28490.128} C_VEL
LIN {X 0,Y 70.671,Z 440.823,A -85,B 0,C 180,E1 -28496.83,E2 -28496.83} C_VEL
LIN {X 0,Y 66.71,Z 449.982,A -85,B 0,C 180,E1 -28505.066,E2 -28505.066} C_VEL
LIN {X 0,Y 64.139,Z 457.341,A -85,B 0,C 180,E1 -28514.09,E2 -28514.09} C_VEL
LIN {X 0,Y 62.949,Z 463.197,A -85,B 0,C 180,E1 -28523.579,E2 -28523.579} C_VEL
LIN {X 0,Y 62.902,Z 466.37,A -85,B 0,C 180,E1 -28529.989,E2 -28529.989} C_VEL
LIN {X 0,Y 63.128,Z 470.096,A -85,B 0,C 180,E1 -28539.602,E2 -28539.602} C_VEL
LIN {X 0,Y 64.846,Z 472.833,A -85,B 0,C 180,E1 -28548.963,E2 -28548.963} C_VEL
LIN {X 0,Y 66.835,Z 474.169,A -85,B 0,C 180,E1 -28554.862,E2 -28554.862} C_VEL
LIN {X 0,Y 72.653,Z 475.729,A -85,B 0,C 180,E1 -28565.467,E2 -28565.467} C_VEL
LIN {X 0,Y 80.832,Z 475.915,A -85,B 0,C 180,E1 -28574.059,E2 -28574.059} C_VEL
LIN {X 0,Y 90.628,Z 474.7,A -85,B 0,C 180,E1 -28580.835,E2 -28580.835} C_VEL
LIN {X 0,Y 101.421,Z 472.006,A -85,B 0,C 180,E1 -28586.244,E2 -28586.244} C_VEL
LIN {X 0,Y 112.99,Z 467.809,A -85,B 0,C 180,E1 -28590.538,E2 -28590.538} C_VEL
LIN {X 0,Y 122.118,Z 463.55,A -85,B 0,C 180,E1 -28593.116,E2 -28593.116} C_VEL
LIN {X 0,Y 133.137,Z 457.219,A -85,B 0,C 180,E1 -28595.573,E2 -28595.573} C_VEL
LIN {X 0,Y 142.872,Z 450.318,A -85,B 0,C 180,E1 -28597.341,E2 -28597.341} C_VEL
LIN {X 0,Y 146.089,Z 447.756,A -85,B 0,C 180,E1 -28597.852,E2 -28597.852} C_VEL
LIN {X 0,Y 147.404,Z 446.618,A -85,B 0,C 180,E1 -28598.565,E2 -28598.565} C_VEL
LIN {X 0,Y 138.187,Z 453.703,A -85,B 0,C 180,E1 -28600.184,E2 -28600.184} C_VEL
LIN {X 0,Y 132.743,Z 457.308,A -85,B 0,C 180,E1 -28601.28,E2 -28601.28} C_VEL
LIN {X 0,Y 127.866,Z 460.209,A -85,B 0,C 180,E1 -28602.035,E2 -28602.035} C_VEL
LIN {X 0,Y 119.072,Z 464.637,A -85,B 0,C 180,E1 -28602.657,E2 -28602.657} C_VEL
LIN {X 0,Y 110.045,Z 468.328,A -85,B 0,C 180,E1 -28603.469,E2 -28603.469} C_VEL
LIN {X 0,Y 104.864,Z 470.058,A -85,B 0,C 180,E1 -28604.633,E2 -28604.633} C_VEL
LIN {X 0,Y 93.032,Z 473.187,A -85,B 0,C 180,E1 -28609.09,E2 -28609.09} C_VEL
LIN {X 0,Y 81.773,Z 474.807,A -85,B 0,C 180,E1 -28615.037,E2 -28615.037} C_VEL
LIN {X 0,Y 74.967,Z 475.092,A -85,B 0,C 180,E1 -28619.965,E2 -28619.965} C_VEL
LIN {X 0,Y 68.92,Z 474.682,A -85,B 0,C 180,E1 -28625.814,E2 -28625.814} C_VEL
LIN {X 0,Y 63.754,Z 473.667,A -85,B 0,C 180,E1 -28632.693,E2 -28632.693} C_VEL
LIN {X 0,Y 58.062,Z 470.85,A -85,B 0,C 180,E1 -28645.013,E2 -28645.013} C_VEL
LIN {X 0,Y 55.884,Z 468.078,A -85,B 0,C 180,E1 -28654.402,E2 -28654.402} C_VEL
LIN {X 0,Y 55.075,Z 464.057,A -85,B 0,C 180,E1 -28665.339,E2 -28665.339} C_VEL
LIN {X 0,Y 55.756,Z 459.328,A -85,B 0,C 180,E1 -28675.459,E2 -28675.459} C_VEL
LIN {X 0,Y 58.055,Z 452.208,A -85,B 0,C 180,E1 -28686.845,E2 -28686.845} C_VEL
LIN {X 0,Y 60.947,Z 445.41,A -85,B 0,C 180,E1 -28694.974,E2 -28694.974} C_VEL
LIN {X 0,Y 64.892,Z 436.978,A -85,B 0,C 180,E1 -28702.494,E2 -28702.494} C_VEL
LIN {X 0,Y 69.295,Z 427.642,A -85,B 0,C 180,E1 -28708.56,E2 -28708.56} C_VEL
LIN {X 0,Y 73.914,Z 417.259,A -85,B 0,C 180,E1 -28713.416,E2 -28713.416} C_VEL
LIN {X 0,Y 78.195,Z 406.24,A -85,B 0,C 180,E1 -28717.102,E2 -28717.102} C_VEL
LIN {X 0,Y 82.262,Z 393.614,A -85,B 0,C 180,E1 -28720.095,E2 -28720.095} C_VEL
LIN {X 0,Y 85.313,Z 381.206,A -85,B 0,C 180,E1 -28722.136,E2 -28722.136} C_VEL
LIN {X 0,Y 87.812,Z 367.075,A -85,B 0,C 180,E1 -28723.527,E2 -28723.527} C_VEL
LIN {X 0,Y 91.488,Z 334.604,A -85,B 0,C 180,E1 -28725.835,E2 -28725.835} C_VEL
LIN {X 0,Y 87.731,Z 324.207,A -85,B 0,C 180,E1 -28729.667,E2 -28729.667} C_VEL
LIN {X 0,Y 83.053,Z 314.453,A -85,B 0,C 180,E1 -28734.863,E2 -28734.863} C_VEL
LIN {X 0,Y 78.915,Z 307.349,A -85,B 0,C 180,E1 -28740.073,E2 -28740.073} C_VEL
LIN {X 0,Y 76.281,Z 303.123,A -85,B 0,C 180,E1 -28744.052,E2 -28744.052} C_VEL
LIN {X 0,Y 74.629,Z 300.476,A -85,B 0,C 180,E1 -28746.94,E2 -28746.94} C_VEL
LIN {X 0,Y 72.319,Z 296.902,A -85,B 0,C 180,E1 -28751.585,E2 -28751.585} C_VEL
LIN {X 0,Y 69.82,Z 294.175,A -85,B 0,C 180,E1 -28757.737,E2 -28757.737} C_VEL
LIN {X 0,Y 68.674,Z 291.666,A -85,B 0,C 180,E1 -28762.17,E2 -28762.17} C_VEL
LIN {X 0,Y 66.596,Z 290.385,A -85,B 0,C 180,E1 -28775.077,E2 -28775.077} C_VEL
LIN {X 0,Y 67.256,Z 290.562,A -85,B 0,C 180,E1 -28786.947,E2 -28786.947} C_VEL
LIN {X 0,Y 69.662,Z 291.835,A -85,B 0,C 180,E1 -28796.586,E2 -28796.586} C_VEL
LIN {X 0,Y 71.071,Z 294.81,A -85,B 0,C 180,E1 -28801.1,E2 -28801.1} C_VEL
LIN {X 0,Y 72.568,Z 296.688,A -85,B 0,C 180,E1 -28804.549,E2 -28804.549} C_VEL
LIN {X 0,Y 74.868,Z 300.346,A -85,B 0,C 180,E1 -28809.15,E2 -28809.15} C_VEL
LIN {X 0,Y 78.257,Z 306.271,A -85,B 0,C 180,E1 -28814.766,E2 -28814.766} C_VEL
LIN {X 0,Y 81.338,Z 311.798,A -85,B 0,C 180,E1 -28818.929,E2 -28818.929} C_VEL
LIN {X 0,Y 85.041,Z 319.495,A -85,B 0,C 180,E1 -28823.407,E2 -28823.407} C_VEL
LIN {X 0,Y 88.998,Z 329.261,A -85,B 0,C 180,E1 -28827.683,E2 -28827.683} C_VEL
LIN {X 0,Y 91.322,Z 338.058,A -85,B 0,C 180,E1 -28830.299,E2 -28830.299} C_VEL
LIN {X 0,Y 87.759,Z 369.197,A -85,B 0,C 180,E1 -28832.505,E2 -28832.505} C_VEL
LIN {X 0,Y 85.349,Z 383.192,A -85,B 0,C 180,E1 -28833.935,E2 -28833.935} C_VEL
LIN {X 0,Y 82.069,Z 396.144,A -85,B 0,C 180,E1 -28836.068,E2 -28836.068} C_VEL
LIN {X 0,Y 77.984,Z 408.306,A -85,B 0,C 180,E1 -28838.928,E2 -28838.928} C_VEL
LIN {X 0,Y 73.321,Z 420.183,A -85,B 0,C 180,E1 -28843.027,E2 -28843.027} C_VEL
LIN {X 0,Y 68.574,Z 430.762,A -85,B 0,C 180,E1 -28848.215,E2 -28848.215} C_VEL
LIN {X 0,Y 64.001,Z 440.337,A -85,B 0,C 180,E1 -28854.782,E2 -28854.782} C_VEL
LIN {X 0,Y 60.364,Z 448.21,A -85,B 0,C 180,E1 -28862.232,E2 -28862.232} C_VEL
LIN {X 0,Y 57.373,Z 455.876,A -85,B 0,C 180,E1 -28872.155,E2 -28872.155} C_VEL
LIN {X 0,Y 55.945,Z 461.991,A -85,B 0,C 180,E1 -28882.771,E2 -28882.771} C_VEL
LIN {X 0,Y 55.87,Z 465.338,A -85,B 0,C 180,E1 -28889.988,E2 -28889.988} C_VEL
LIN {X 0,Y 56.187,Z 469.225,A -85,B 0,C 180,E1 -28900.802,E2 -28900.802} C_VEL
LIN {X 0,Y 58.202,Z 472.144,A -85,B 0,C 180,E1 -28911.226,E2 -28911.226} C_VEL
LIN {X 0,Y 63.353,Z 474.706,A -85,B 0,C 180,E1 -28923.674,E2 -28923.674} C_VEL
LIN {X 0,Y 71.231,Z 475.842,A -85,B 0,C 180,E1 -28933.668,E2 -28933.668} C_VEL
LIN {X 0,Y 80.948,Z 475.56,A -85,B 0,C 180,E1 -28941.373,E2 -28941.373} C_VEL
LIN {X 0,Y 91.926,Z 473.89,A -85,B 0,C 180,E1 -28947.229,E2 -28947.229} C_VEL
LIN {X 0,Y 98.328,Z 472.35,A -85,B 0,C 180,E1 -28949.95,E2 -28949.95} C_VEL
LIN {X 0,Y 109.706,Z 468.636,A -85,B 0,C 180,E1 -28953.734,E2 -28953.734} C_VEL
LIN {X 0,Y 119.113,Z 464.648,A -85,B 0,C 180,E1 -28956.125,E2 -28956.125} C_VEL
LIN {X 0,Y 128.774,Z 459.595,A -85,B 0,C 180,E1 -28958.077,E2 -28958.077} C_VEL
LIN {X 0,Y 128.077,Z 459.985,A -85,B 0,C 180,E1 -28958.866,E2 -28958.866} C_VEL
LIN {X 0,Y 116.828,Z 465.56,A -85,B 0,C 180,E1 -28961.294,E2 -28961.294} C_VEL
LIN {X 0,Y 104.864,Z 470.058,A -85,B 0,C 180,E1 -28964.633,E2 -28964.633} C_VEL
LIN {X 0,Y 99.651,Z 471.594,A -85,B 0,C 180,E1 -28965.97,E2 -28965.97} C_VEL
LIN {X 0,Y 90.305,Z 473.596,A -85,B 0,C 180,E1 -28967.575,E2 -28967.575} C_VEL
LIN {X 0,Y 81.008,Z 474.822,A -85,B 0,C 180,E1 -28969.638,E2 -28969.638} C_VEL
LIN {X 0,Y 75.99,Z 475.086,A -85,B 0,C 180,E1 -28971.862,E2 -28971.862} C_VEL
LIN {X 0,Y 70.476,Z 475.149,A -85,B 0,C 180,E1 -28975.588,E2 -28975.588} C_VEL
LIN {X 0,Y 63.28,Z 474.539,A -85,B 0,C 180,E1 -28982.073,E2 -28982.073} C_VEL
LIN {X 0,Y 57.103,Z 473.127,A -85,B 0,C 180,E1 -28990.139,E2 -28990.139} C_VEL
LIN {X 0,Y 50.81,Z 469.728,A -85,B 0,C 180,E1 -29004.457,E2 -29004.457} C_VEL
LIN {X 0,Y 48.215,Z 465.286,A -85,B 0,C 180,E1 -29019.137,E2 -29019.137} C_VEL
LIN {X 0,Y 48.231,Z 460.849,A -85,B 0,C 180,E1 -29030.819,E2 -29030.819} C_VEL
LIN {X 0,Y 49.679,Z 455.319,A -85,B 0,C 180,E1 -29042.195,E2 -29042.195} C_VEL
LIN {X 0,Y 52.598,Z 448.353,A -85,B 0,C 180,E1 -29052.939,E2 -29052.939} C_VEL
LIN {X 0,Y 57.059,Z 439.275,A -85,B 0,C 180,E1 -29062.937,E2 -29062.937} C_VEL
LIN {X 0,Y 61.845,Z 429.893,A -85,B 0,C 180,E1 -29070.011,E2 -29070.011} C_VEL
LIN {X 0,Y 67.385,Z 418.362,A -85,B 0,C 180,E1 -29075.997,E2 -29075.997} C_VEL
LIN {X 0,Y 72.071,Z 407.231,A -85,B 0,C 180,E1 -29079.962,E2 -29079.962} C_VEL
LIN {X 0,Y 76.263,Z 395.073,A -85,B 0,C 180,E1 -29082.99,E2 -29082.99} C_VEL
LIN {X 0,Y 79.775,Z 381.863,A -85,B 0,C 180,E1 -29085.252,E2 -29085.252} C_VEL
LIN {X 0,Y 82.393,Z 367.964,A -85,B 0,C 180,E1 -29086.65,E2 -29086.65} C_VEL
LIN {X 0,Y 86.137,Z 337.538,A -85,B 0,C 180,E1 -29088.761,E2 -29088.761} C_VEL
LIN {X 0,Y 85.86,Z 335.747,A -85,B 0,C 180,E1 -29089.221,E2 -29089.221} C_VEL
LIN {X 0,Y 83.239,Z 327.974,A -85,B 0,C 180,E1 -29092.401,E2 -29092.401} C_VEL
LIN {X 0,Y 79.283,Z 319.358,A -85,B 0,C 180,E1 -29097.351,E2 -29097.351} C_VEL
LIN {X 0,Y 75.732,Z 312.797,A -85,B 0,C 180,E1 -29102.512,E2 -29102.512} C_VEL
LIN {X 0,Y 73.322,Z 308.562,A -85,B 0,C 180,E1 -29106.754,E2 -29106.754} C_VEL
LIN {X 0,Y 72.065,Z 306.47,A -85,B 0,C 180,E1 -29109.215,E2 -29109.215} C_VEL
LIN {X 0,Y 69.887,Z 303.065,A -85,B 0,C 180,E1 -29114.197,E2 -29114.197} C_VEL
LIN {X 0,Y 67.883,Z 300.31,A -85,B 0,C 180,E1 -29120.283,E2 -29120.283} C_VEL
LIN {X 0,Y 67.22,Z 298.526,A -85,B 0,C 180,E1 -29123.337,E2 -29123.337} C_VEL
LIN {X 0,Y 65.516,Z 297.413,A -85,B 0,C 180,E1 -29134.637,E2 -29134.637} C_VEL
LIN {X 0,Y 65.943,Z 297.469,A -85,B 0,C 180,E1 -29145.625,E2 -29145.625} C_VEL
LIN {X 0,Y 67.952,Z 298.603,A -85,B 0,C 180,E1 -29154.883,E2 -29154.883} C_VEL
LIN {X 0,Y 69.636,Z 301.959,A -85,B 0,C 180,E1 -29160.629,E2 -29160.629} C_VEL
LIN {X 0,Y 70.509,Z 303.357,A -85,B 0,C 180,E1 -29162.894,E2 -29162.894} C_VEL
LIN {X 0,Y 72.926,Z 307.573,A -85,B 0,C 180,E1 -29168.173,E2 -29168.173} C_VEL
LIN {X 0,Y 76.135,Z 313.484,A -85,B 0,C 180,E1 -29173.9,E2 -29173.9} C_VEL
LIN {X 0,Y 79.932,Z 321.474,A -85,B 0,C 180,E1 -29179.415,E2 -29179.415} C_VEL
LIN {X 0,Y 84.045,Z 331.801,A -85,B 0,C 180,E1 -29184.624,E2 -29184.624} C_VEL
LIN {X 0,Y 86.014,Z 339.586,A -85,B 0,C 180,E1 -29187.229,E2 -29187.229} C_VEL
LIN {X 0,Y 82.599,Z 368.106,A -85,B 0,C 180,E1 -29189.252,E2 -29189.252} C_VEL
LIN {X 0,Y 80.162,Z 382.046,A -85,B 0,C 180,E1 -29190.636,E2 -29190.636} C_VEL
LIN {X 0,Y 76.749,Z 395.126,A -85,B 0,C 180,E1 -29192.706,E2 -29192.706} C_VEL
LIN {X 0,Y 72.32,Z 407.855,A -85,B 0,C 180,E1 -29195.709,E2 -29195.709} C_VEL
LIN {X 0,Y 67.479,Z 419.541,A -85,B 0,C 180,E1 -29199.8,E2 -29199.8} C_VEL
LIN {X 0,Y 62.383,Z 430.207,A -85,B 0,C 180,E1 -29205.227,E2 -29205.227} C_VEL
LIN {X 0,Y 57.45,Z 439.856,A -85,B 0,C 180,E1 -29212.275,E2 -29212.275} C_VEL
LIN {X 0,Y 53.495,Z 447.787,A -85,B 0,C 180,E1 -29220.47,E2 -29220.47} C_VEL
LIN {X 0,Y 50.262,Z 455.489,A -85,B 0,C 180,E1 -29231.648,E2 -29231.648} C_VEL
LIN {X 0,Y 48.962,Z 460.718,A -85,B 0,C 180,E1 -29241.733,E2 -29241.733} C_VEL
LIN {X 0,Y 48.839,Z 464.186,A -85,B 0,C 180,E1 -29249.986,E2 -29249.986} C_VEL
LIN {X 0,Y 49.013,Z 467.059,A -85,B 0,C 180,E1 -29258.23,E2 -29258.23} C_VEL
LIN {X 0,Y 51.674,Z 471.454,A -85,B 0,C 180,E1 -29274.065,E2 -29274.065} C_VEL
LIN {X 0,Y 57.573,Z 474.218,A -85,B 0,C 180,E1 -29287.599,E2 -29287.599} C_VEL
LIN {X 0,Y 66.28,Z 475.609,A -85,B 0,C 180,E1 -29297.907,E2 -29297.907} C_VEL
LIN {X 0,Y 76.723,Z 475.626,A -85,B 0,C 180,E1 -29305.513,E2 -29305.513} C_VEL
LIN {X 0,Y 88.291,Z 474.208,A -85,B 0,C 180,E1 -29311.1,E2 -29311.1} C_VEL
LIN {X 0,Y 100.49,Z 471.391,A -85,B 0,C 180,E1 -29315.375,E2 -29315.375} C_VEL
LIN {X 0,Y 108.292,Z 468.9,A -85,B 0,C 180,E1 -29317.492,E2 -29317.492} C_VEL
LIN {X 0,Y 110.697,Z 467.983,A -85,B 0,C 180,E1 -29318.874,E2 -29318.874} C_VEL
LIN {X 0,Y 100.22,Z 471.32,A -85,B 0,C 180,E1 -29321.576,E2 -29321.576} C_VEL
LIN {X 0,Y 86.769,Z 474.148,A -85,B 0,C 180,E1 -29326.361,E2 -29326.361} C_VEL
LIN {X 0,Y 75.99,Z 475.086,A -85,B 0,C 180,E1 -29331.862,E2 -29331.862} C_VEL
LIN {X 0,Y 71.059,Z 475.191,A -85,B 0,C 180,E1 -29334.416,E2 -29334.416} C_VEL
LIN {X 0,Y 62.158,Z 474.678,A -85,B 0,C 180,E1 -29338.205,E2 -29338.205} C_VEL
LIN {X 0,Y 53.773,Z 473.325,A -85,B 0,C 180,E1 -29343.283,E2 -29343.283} C_VEL
LIN {X 0,Y 49.912,Z 472.191,A -85,B 0,C 180,E1 -29348.071,E2 -29348.071} C_VEL
LIN {X 0,Y 43.425,Z 468.26,A -85,B 0,C 180,E1 -29364.266,E2 -29364.266} C_VEL
LIN {X 0,Y 41.29,Z 464.566,A -85,B 0,C 180,E1 -29377.51,E2 -29377.51} C_VEL
LIN {X 0,Y 41.298,Z 459.425,A -85,B 0,C 180,E1 -29392.503,E2 -29392.503} C_VEL
LIN {X 0,Y 43.196,Z 453.327,A -85,B 0,C 180,E1 -29406.022,E2 -29406.022} C_VEL
LIN {X 0,Y 46.367,Z 446.673,A -85,B 0,C 180,E1 -29416.874,E2 -29416.874} C_VEL
LIN {X 0,Y 51.167,Z 437.739,A -85,B 0,C 180,E1 -29427.061,E2 -29427.061} C_VEL
LIN {X 0,Y 56.781,Z 427.611,A -85,B 0,C 180,E1 -29434.752,E2 -29434.752} C_VEL
LIN {X 0,Y 61.796,Z 417.762,A -85,B 0,C 180,E1 -29439.837,E2 -29439.837} C_VEL
LIN {X 0,Y 67.062,Z 405.797,A -85,B 0,C 180,E1 -29444.036,E2 -29444.036} C_VEL
LIN {X 0,Y 71.677,Z 392.845,A -85,B 0,C 180,E1 -29447.117,E2 -29447.117} C_VEL
LIN {X 0,Y 75.149,Z 379.66,A -85,B 0,C 180,E1 -29449.174,E2 -29449.174} C_VEL
LIN {X 0,Y 77.707,Z 366.03,A -85,B 0,C 180,E1 -29450.39,E2 -29450.39} C_VEL
LIN {X 0,Y 81.089,Z 338.598,A -85,B 0,C 180,E1 -29452.35,E2 -29452.35} C_VEL
LIN {X 0,Y 79.06,Z 332.218,A -85,B 0,C 180,E1 -29455.179,E2 -29455.179} C_VEL
LIN {X 0,Y 75.675,Z 324.295,A -85,B 0,C 180,E1 -29460.063,E2 -29460.063} C_VEL
LIN {X 0,Y 72.683,Z 318.197,A -85,B 0,C 180,E1 -29465.19,E2 -29465.19} C_VEL
LIN {X 0,Y 69.941,Z 312.913,A -85,B 0,C 180,E1 -29470.872,E2 -29470.872} C_VEL
LIN {X 0,Y 67.924,Z 309.527,A -85,B 0,C 180,E1 -29476.12,E2 -29476.12} C_VEL
LIN {X 0,Y 66.105,Z 306.584,A -85,B 0,C 180,E1 -29482.682,E2 -29482.682} C_VEL
LIN {X 0,Y 65.64,Z 305.322,A -85,B 0,C 180,E1 -29485.182,E2 -29485.182} C_VEL
LIN {X 0,Y 64.43,Z 304.471,A -85,B 0,C 180,E1 -29494.178,E2 -29494.178} C_VEL
LIN {X 0,Y 64.986,Z 304.557,A -85,B 0,C 180,E1 -29506.777,E2 -29506.777} C_VEL
LIN {X 0,Y 66.369,Z 305.503,A -85,B 0,C 180,E1 -29513.39,E2 -29513.39} C_VEL
LIN {X 0,Y 68.351,Z 309.57,A -85,B 0,C 180,E1 -29520.641,E2 -29520.641} C_VEL
LIN {X 0,Y 70.512,Z 313.781,A -85,B 0,C 180,E1 -29526.12,E2 -29526.12} C_VEL
LIN {X 0,Y 73.522,Z 319.977,A -85,B 0,C 180,E1 -29532.166,E2 -29532.166} C_VEL
LIN {X 0,Y 76.627,Z 327.298,A -85,B 0,C 180,E1 -29537.338,E2 -29537.338} C_VEL
LIN {X 0,Y 80.013,Z 336.695,A -85,B 0,C 180,E1 -29542.202,E2 -29542.202} C_VEL
LIN {X 0,Y 81.014,Z 341.279,A -85,B 0,C 180,E1 -29543.825,E2 -29543.825} C_VEL
LIN {X 0,Y 76.811,Z 373.004,A -85,B 0,C 180,E1 -29546.037,E2 -29546.037} C_VEL
LIN {X 0,Y 74.061,Z 385.851,A -85,B 0,C 180,E1 -29547.523,E2 -29547.523} C_VEL
LIN {X 0,Y 70.159,Z 398.945,A -85,B 0,C 180,E1 -29549.857,E2 -29549.857} C_VEL
LIN {X 0,Y 65.164,Z 411.605,A -85,B 0,C 180,E1 -29553.278,E2 -29553.278} C_VEL
LIN {X 0,Y 60.015,Z 422.657,A -85,B 0,C 180,E1 -29557.754,E2 -29557.754} C_VEL
LIN {X 0,Y 54.702,Z 432.713,A -85,B 0,C 180,E1 -29563.706,E2 -29563.706} C_VEL
LIN {X 0,Y 49.168,Z 442.622,A -85,B 0,C 180,E1 -29572.575,E2 -29572.575} C_VEL
LIN {X 0,Y 44.682,Z 451.357,A -85,B 0,C 180,E1 -29584.354,E2 -29584.354} C_VEL
LIN {X 0,Y 42.198,Z 458.306,A -85,B 0,C 180,E1 -29597.967,E2 -29597.967} C_VEL
LIN {X 0,Y 41.809,Z 462.996,A -85,B 0,C 180,E1 -29609.984,E2 -29609.984} C_VEL
LIN {X 0,Y 42.066,Z 466.027,A -85,B 0,C 180,E1 -29619.601,E2 -29619.601} C_VEL
LIN {X 0,Y 45.313,Z 470.638,A -85,B 0,C 180,E1 -29637.712,E2 -29637.712} C_VEL
LIN {X 0,Y 52.125,Z 473.705,A -85,B 0,C 180,E1 -29652.369,E2 -29652.369} C_VEL
LIN {X 0,Y 61.749,Z 475.339,A -85,B 0,C 180,E1 -29662.797,E2 -29662.797} C_VEL
LIN {X 0,Y 72.944,Z 475.596,A -85,B 0,C 180,E1 -29670.106,E2 -29670.106} C_VEL
LIN {X 0,Y 85.085,Z 474.497,A -85,B 0,C 180,E1 -29675.291,E2 -29675.291} C_VEL
LIN {X 0,Y 91.354,Z 473.424,A -85,B 0,C 180,E1 -29677.374,E2 -29677.374} C_VEL
LIN {X 0,Y 93.913,Z 472.847,A -85,B 0,C 180,E1 -29678.755,E2 -29678.755} C_VEL
LIN {X 0,Y 86.61,Z 474.154,A -85,B 0,C 180,E1 -29681.029,E2 -29681.029} C_VEL
LIN {X 0,Y 78.145,Z 475.049,A -85,B 0,C 180,E1 -29684.313,E2 -29684.313} C_VEL
LIN {X 0,Y 70.081,Z 475.321,A -85,B 0,C 180,E1 -29688.392,E2 -29688.392} C_VEL
LIN {X 0,Y 62.606,Z 474.904,A -85,B 0,C 180,E1 -29693.512,E2 -29693.512} C_VEL
LIN {X 0,Y 55.789,Z 473.881,A -85,B 0,C 180,E1 -29699.953,E2 -29699.953} C_VEL
LIN {X 0,Y 49.912,Z 472.191,A -85,B 0,C 180,E1 -29708.071,E2 -29708.071} C_VEL
LIN {X 0,Y 47.696,Z 471.327,A -85,B 0,C 180,E1 -29711.742,E2 -29711.742} C_VEL
LIN {X 0,Y 43.972,Z 469.718,A -85,B 0,C 180,E1 -29717.135,E2 -29717.135} C_VEL
LIN {X 0,Y 35.905,Z 464.828,A -85,B 0,C 180,E1 -29732.013,E2 -29732.013} C_VEL
LIN {X 0,Y 34.154,Z 462.311,A -85,B 0,C 180,E1 -29740.426,E2 -29740.426} C_VEL
LIN {X 0,Y 34.005,Z 461.397,A -85,B 0,C 180,E1 -29743.444,E2 -29743.444} C_VEL
LIN {X 0,Y 35.08,Z 455.541,A -85,B 0,C 180,E1 -29761.079,E2 -29761.079} C_VEL
LIN {X 0,Y 38.617,Z 448.061,A -85,B 0,C 180,E1 -29776.925,E2 -29776.925} C_VEL
LIN {X 0,Y 43.251,Z 440.154,A -85,B 0,C 180,E1 -29788.068,E2 -29788.068} C_VEL
LIN {X 0,Y 48.523,Z 431.475,A -85,B 0,C 180,E1 -29796.183,E2 -29796.183} C_VEL
LIN {X 0,Y 54.843,Z 420.203,A -85,B 0,C 180,E1 -29802.972,E2 -29802.972} C_VEL
LIN {X 0,Y 60.067,Z 409.631,A -85,B 0,C 180,E1 -29807.113,E2 -29807.113} C_VEL
LIN {X 0,Y 64.804,Z 398.095,A -85,B 0,C 180,E1 -29810.215,E2 -29810.215} C_VEL
LIN {X 0,Y 69.054,Z 384.694,A -85,B 0,C 180,E1 -29812.565,E2 -29812.565} C_VEL
LIN {X 0,Y 72.043,Z 371.44,A -85,B 0,C 180,E1 -29814.049,E2 -29814.049} C_VEL
LIN {X 0,Y 76.226,Z 341.822,A -85,B 0,C 180,E1 -29815.986,E2 -29815.986} C_VEL
LIN {X 0,Y 76.129,Z 340.192,A -85,B 0,C 180,E1 -29816.389,E2 -29816.389} C_VEL
LIN {X 0,Y 74.975,Z 336.274,A -85,B 0,C 180,E1 -29818.32,E2 -29818.32} C_VEL
LIN {X 0,Y 72.108,Z 328.798,A -85,B 0,C 180,E1 -29823.335,E2 -29823.335} C_VEL
LIN {X 0,Y 69.411,Z 322.849,A -85,B 0,C 180,E1 -29828.813,E2 -29828.813} C_VEL
LIN {X 0,Y 67.318,Z 318.515,A -85,B 0,C 180,E1 -29834.074,E2 -29834.074} C_VEL
LIN {X 0,Y 65.948,Z 315.916,A -85,B 0,C 180,E1 -29838.447,E2 -29838.447} C_VEL
LIN {X 0,Y 64.16,Z 312.168,A -85,B 0,C 180,E1 -29846.843,E2 -29846.843} C_VEL
LIN {X 0,Y 63.339,Z 311.52,A -85,B 0,C 180,E1 -29853.7,E2 -29853.7} C_VEL
LIN {X 0,Y 63.699,Z 311.503,A -85,B 0,C 180,E1 -29865.611,E2 -29865.611} C_VEL
LIN {X 0,Y 64.821,Z 312.381,A -85,B 0,C 180,E1 -29871.861,E2 -29871.861} C_VEL
LIN {X 0,Y 66.398,Z 316.044,A -85,B 0,C 180,E1 -29878.597,E2 -29878.597} C_VEL
LIN {X 0,Y 68.403,Z 320.498,A -85,B 0,C 180,E1 -29884.507,E2 -29884.507} C_VEL
LIN {X 0,Y 70.983,Z 326.468,A -85,B 0,C 180,E1 -29890.31,E2 -29890.31} C_VEL
LIN {X 0,Y 73.562,Z 333.542,A -85,B 0,C 180,E1 -29895.32,E2 -29895.32} C_VEL
LIN {X 0,Y 75.892,Z 341.106,A -85,B 0,C 180,E1 -29899.324,E2 -29899.324} C_VEL
LIN {X 0,Y 76.217,Z 342.864,A -85,B 0,C 180,E1 -29899.97,E2 -29899.97} C_VEL
LIN {X 0,Y 72.044,Z 372.857,A -85,B 0,C 180,E1 -29902.004,E2 -29902.004} C_VEL
LIN {X 0,Y 68.978,Z 386.248,A -85,B 0,C 180,E1 -29903.487,E2 -29903.487} C_VEL
LIN {X 0,Y 65.062,Z 398.713,A -85,B 0,C 180,E1 -29905.686,E2 -29905.686} C_VEL
LIN {X 0,Y 60.131,Z 410.614,A -85,B 0,C 180,E1 -29908.778,E2 -29908.778} C_VEL
LIN {X 0,Y 53.958,Z 423.062,A -85,B 0,C 180,E1 -29913.844,E2 -29913.844} C_VEL
LIN {X 0,Y 48.244,Z 432.99,A -85,B 0,C 180,E1 -29920.09,E2 -29920.09} C_VEL
LIN {X 0,Y 42.755,Z 442.025,A -85,B 0,C 180,E1 -29928.869,E2 -29928.869} C_VEL
LIN {X 0,Y 37.769,Z 450.839,A -85,B 0,C 180,E1 -29942.257,E2 -29942.257} C_VEL
LIN {X 0,Y 35.088,Z 457.881,A -85,B 0,C 180,E1 -29958.426,E2 -29958.426} C_VEL
LIN {X 0,Y 34.924,Z 463.384,A -85,B 0,C 180,E1 -29975.755,E2 -29975.755} C_VEL
LIN {X 0,Y 37.758,Z 468.703,A -85,B 0,C 180,E1 -29997.71,E2 -29997.71} C_VEL
LIN {X 0,Y 42.799,Z 471.626,A -85,B 0,C 180,E1 -30011.037,E2 -30011.037} C_VEL
LIN {X 0,Y 47.128,Z 473.093,A -85,B 0,C 180,E1 -30018.19,E2 -30018.19} C_VEL
LIN {X 0,Y 57.738,Z 475.009,A -85,B 0,C 180,E1 -30028.411,E2 -30028.411} C_VEL
LIN {X 0,Y 63.553,Z 475.459,A -85,B 0,C 180,E1 -30032.188,E2 -30032.188} C_VEL
LIN {X 0,Y 75.968,Z 475.299,A -85,B 0,C 180,E1 -30037.662,E2 -30037.662} C_VEL
LIN {X 0,Y 77.434,Z 475.175,A -85,B 0,C 180,E1 -30038.677,E2 -30038.677} C_VEL
LIN {X 0,Y 65.948,Z 475.342,A -85,B 0,C 180,E1 -30043.521,E2 -30043.521} C_VEL
LIN {X 0,Y 57.282,Z 474.626,A -85,B 0,C 180,E1 -30048.904,E2 -30048.904} C_VEL
LIN {X 0,Y 46.274,Z 472.301,A -85,B 0,C 180,E1 -30059.943,E2 -30059.943} C_VEL
LIN {X 0,Y 38.781,Z 468.914,A -85,B 0,C 180,E1 -30074.384,E2 -30074.384} C_VEL
LIN {X 0,Y 35.21,Z 465.374,A -85,B 0,C 180,E1 -30088.745,E2 -30088.745} C_VEL
LIN {X 0,Y 34.005,Z 461.397,A -85,B 0,C 180,E1 -30103.444,E2 -30103.444} C_VEL
LIN {X 0,Y 33.571,Z 458.638,A -85,B 0,C 180,E1 -30112.239,E2 -30112.239} C_VEL
LIN {X 0,Y 32.784,Z 455.529,A -85,B 0,C 180,E1 -30120.906,E2 -30120.906} C_VEL
LIN {X 0,Y 32.703,Z 447.31,A -85,B 0,C 180,E1 -30140.932,E2 -30140.932} C_VEL
LIN {X 0,Y 34.617,Z 443.395,A -85,B 0,C 180,E1 -30148.003,E2 -30148.003} C_VEL
LIN {X 0,Y 40.653,Z 434.436,A -85,B 0,C 180,E1 -30158.717,E2 -30158.717} C_VEL
LIN {X 0,Y 47.253,Z 424.036,A -85,B 0,C 180,E1 -30166.208,E2 -30166.208} C_VEL
LIN {X 0,Y 53.018,Z 413.752,A -85,B 0,C 180,E1 -30170.795,E2 -30170.795} C_VEL
LIN {X 0,Y 58.655,Z 401.56,A -85,B 0,C 180,E1 -30174.339,E2 -30174.339} C_VEL
LIN {X 0,Y 63.359,Z 388.651,A -85,B 0,C 180,E1 -30176.725,E2 -30176.725} C_VEL
LIN {X 0,Y 66.757,Z 375.768,A -85,B 0,C 180,E1 -30178.275,E2 -30178.275} C_VEL
LIN {X 0,Y 69.742,Z 358.232,A -85,B 0,C 180,E1 -30179.381,E2 -30179.381} C_VEL
LIN {X 0,Y 71.834,Z 342.713,A -85,B 0,C 180,E1 -30180.422,E2 -30180.422} C_VEL
LIN {X 0,Y 69.387,Z 334.96,A -85,B 0,C 180,E1 -30185.547,E2 -30185.547} C_VEL
LIN {X 0,Y 67.042,Z 329.135,A -85,B 0,C 180,E1 -30190.989,E2 -30190.989} C_VEL
LIN {X 0,Y 65.113,Z 324.466,A -85,B 0,C 180,E1 -30196.868,E2 -30196.868} C_VEL
LIN {X 0,Y 64.048,Z 322.192,A -85,B 0,C 180,E1 -30201.052,E2 -30201.052} C_VEL
LIN {X 0,Y 62.777,Z 319.031,A -85,B 0,C 180,E1 -30208.325,E2 -30208.325} C_VEL
LIN {X 0,Y 62.17,Z 318.492,A -85,B 0,C 180,E1 -30214.761,E2 -30214.761} C_VEL
LIN {X 0,Y 62.545,Z 318.503,A -85,B 0,C 180,E1 -30225.339,E2 -30225.339} C_VEL
LIN {X 0,Y 63.302,Z 319.133,A -85,B 0,C 180,E1 -30230.158,E2 -30230.158} C_VEL
LIN {X 0,Y 64.453,Z 322.235,A -85,B 0,C 180,E1 -30236.042,E2 -30236.042} C_VEL
LIN {X 0,Y 66.135,Z 326.655,A -85,B 0,C 180,E1 -30242.141,E2 -30242.141} C_VEL
LIN {X 0,Y 68.182,Z 332.336,A -85,B 0,C 180,E1 -30247.693,E2 -30247.693} C_VEL
LIN {X 0,Y 70.185,Z 338.553,A -85,B 0,C 180,E1 -30252.288,E2 -30252.288} C_VEL
LIN {X 0,Y 71.753,Z 344.334,A -85,B 0,C 180,E1 -30255.618,E2 -30255.618} C_VEL
LIN {X 0,Y 68.699,Z 366.504,A -85,B 0,C 180,E1 -30257.053,E2 -30257.053} C_VEL
LIN {X 0,Y 65.939,Z 380.601,A -85,B 0,C 180,E1 -30258.199,E2 -30258.199} C_VEL
LIN {X 0,Y 62.141,Z 393.605,A -85,B 0,C 180,E1 -30259.953,E2 -30259.953} C_VEL
LIN {X 0,Y 57.614,Z 405.047,A -85,B 0,C 180,E1 -30262.254,E2 -30262.254} C_VEL
LIN {X 0,Y 51.83,Z 416.951,A -85,B 0,C 180,E1 -30266.032,E2 -30266.032} C_VEL
LIN {X 0,Y 45.392,Z 428.064,A -85,B 0,C 180,E1 -30271.591,E2 -30271.591} C_VEL
LIN {X 0,Y 38.914,Z 437.949,A -85,B 0,C 180,E1 -30279.837,E2 -30279.837} C_VEL
LIN {X 0,Y 32.536,Z 447.516,A -85,B 0,C 180,E1 -30293.532,E2 -30293.532} C_VEL
LIN {X 0,Y 28.586,Z 455.142,A -85,B 0,C 180,E1 -30312.077,E2 -30312.077} C_VEL
LIN {X 0,Y 27.751,Z 460.304,A -85,B 0,C 180,E1 -30329.975,E2 -30329.975} C_VEL
LIN {X 0,Y 28.387,Z 463.657,A -85,B 0,C 180,E1 -30344.309,E2 -30344.309} C_VEL
LIN {X 0,Y 33.484,Z 468.862,A -85,B 0,C 180,E1 -30368.999,E2 -30368.999} C_VEL
LIN {X 0,Y 42.731,Z 472.443,A -85,B 0,C 180,E1 -30385.292,E2 -30385.292} C_VEL
LIN {X 0,Y 54.361,Z 474.608,A -85,B 0,C 180,E1 -30394.789,E2 -30394.789} C_VEL
LIN {X 0,Y 60.567,Z 475.18,A -85,B 0,C 180,E1 -30398.138,E2 -30398.138} C_VEL
LIN {X 0,Y 60.2,Z 475.14,A -85,B 0,C 180,E1 -30399.026,E2 -30399.026} C_VEL
LIN {X 0,Y 51.095,Z 473.992,A -85,B 0,C 180,E1 -30404.279,E2 -30404.279} C_VEL
LIN {X 0,Y 39.78,Z 471.17,A -85,B 0,C 180,E1 -30415.326,E2 -30415.326} C_VEL
LIN {X 0,Y 31.256,Z 467.031,A -85,B 0,C 180,E1 -30432.907,E2 -30432.907} C_VEL
LIN {X 0,Y 27.383,Z 462.179,A -85,B 0,C 180,E1 -30454.583,E2 -30454.583} C_VEL
LIN {X 0,Y 27.377,Z 456.997,A -85,B 0,C 180,E1 -30475.287,E2 -30475.287} C_VEL
LIN {X 0,Y 30.166,Z 450.527,A -85,B 0,C 180,E1 -30494.291,E2 -30494.291} C_VEL
LIN {X 0,Y 34.617,Z 443.395,A -85,B 0,C 180,E1 -30508.003,E2 -30508.003} C_VEL
LIN {X 0,Y 36.763,Z 439.39,A -85,B 0,C 180,E1 -30513.975,E2 -30513.975} C_VEL
LIN {X 0,Y 39.246,Z 432.244,A -85,B 0,C 180,E1 -30523.656,E2 -30523.656} C_VEL
LIN {X 0,Y 42.207,Z 424.586,A -85,B 0,C 180,E1 -30531.647,E2 -30531.647} C_VEL
LIN {X 0,Y 44.836,Z 419.691,A -85,B 0,C 180,E1 -30534.622,E2 -30534.622} C_VEL
LIN {X 0,Y 50.467,Z 409.669,A -85,B 0,C 180,E1 -30538.05,E2 -30538.05} C_VEL
LIN {X 0,Y 56.106,Z 397.245,A -85,B 0,C 180,E1 -30540.839,E2 -30540.839} C_VEL
LIN {X 0,Y 60.815,Z 383.447,A -85,B 0,C 180,E1 -30542.754,E2 -30542.754} C_VEL
LIN {X 0,Y 63.99,Z 369.908,A -85,B 0,C 180,E1 -30543.875,E2 -30543.875} C_VEL
LIN {X 0,Y 67.673,Z 345.904,A -85,B 0,C 180,E1 -30545.122,E2 -30545.122} C_VEL
LIN {X 0,Y 67.648,Z 344.638,A -85,B 0,C 180,E1 -30545.493,E2 -30545.493} C_VEL
LIN {X 0,Y 66,Z 339.054,A -85,B 0,C 180,E1 -30549.723,E2 -30549.723} C_VEL
LIN {X 0,Y 64.023,Z 333.118,A -85,B 0,C 180,E1 -30555.948,E2 -30555.948} C_VEL
LIN {X 0,Y 62.83,Z 329.828,A -85,B 0,C 180,E1 -30560.915,E2 -30560.915} C_VEL
LIN {X 0,Y 61.494,Z 325.958,A -85,B 0,C 180,E1 -30569.405,E2 -30569.405} C_VEL
LIN {X 0,Y 61.022,Z 325.412,A -85,B 0,C 180,E1 -30579.835,E2 -30579.835} C_VEL
LIN {X 0,Y 61.806,Z 325.804,A -85,B 0,C 180,E1 -30588.111,E2 -30588.111} C_VEL
LIN {X 0,Y 62.709,Z 328.732,A -85,B 0,C 180,E1 -30593.855,E2 -30593.855} C_VEL
LIN {X 0,Y 63.92,Z 332.671,A -85,B 0,C 180,E1 -30599.386,E2 -30599.386} C_VEL
LIN {X 0,Y 65.592,Z 338.343,A -85,B 0,C 180,E1 -30605.073,E2 -30605.073} C_VEL
LIN {X 0,Y 67.463,Z 345.554,A -85,B 0,C 180,E1 -30610.243,E2 -30610.243} C_VEL
LIN {X 0,Y 67.691,Z 346.463,A -85,B 0,C 180,E1 -30610.812,E2 -30610.812} C_VEL
LIN {X 0,Y 64.077,Z 370.501,A -85,B 0,C 180,E1 -30612.154,E2 -30612.154} C_VEL
LIN {X 0,Y 61.123,Z 383.421,A -85,B 0,C 180,E1 -30613.186,E2 -30613.186} C_VEL
LIN {X 0,Y 56.702,Z 396.724,A -85,B 0,C 180,E1 -30615.004,E2 -30615.004} C_VEL
LIN {X 0,Y 51.543,Z 408.336,A -85,B 0,C 180,E1 -30617.313,E2 -30617.313} C_VEL
LIN {X 0,Y 45.216,Z 419.896,A -85,B 0,C 180,E1 -30621.119,E2 -30621.119} C_VEL
LIN {X 0,Y 37.671,Z 431.372,A -85,B 0,C 180,E1 -30627.567,E2 -30627.567} C_VEL
LIN {X 0,Y 30.81,Z 440.643,A -85,B 0,C 180,E1 -30636.989,E2 -30636.989} C_VEL
LIN {X 0,Y 24.212,Z 449.593,A -85,B 0,C 180,E1 -30654.477,E2 -30654.477} C_VEL
LIN {X 0,Y 20.882,Z 456.77,A -85,B 0,C 180,E1 -30680.279,E2 -30680.279} C_VEL
LIN {X 0,Y 21.073,Z 460.698,A -85,B 0,C 180,E1 -30699.566,E2 -30699.566} C_VEL
LIN {X 0,Y 24.228,Z 465.329,A -85,B 0,C 180,E1 -30725.427,E2 -30725.427} C_VEL
LIN {X 0,Y 33.453,Z 469.947,A -85,B 0,C 180,E1 -30747.138,E2 -30747.138} C_VEL
LIN {X 0,Y 41.197,Z 472.227,A -85,B 0,C 180,E1 -30755.565,E2 -30755.565} C_VEL
LIN {X 0,Y 44.079,Z 472.826,A -85,B 0,C 180,E1 -30759.313,E2 -30759.313} C_VEL
LIN {X 0,Y 34.342,Z 470.07,A -85,B 0,C 180,E1 -30768.113,E2 -30768.113} C_VEL
LIN {X 0,Y 27.364,Z 467.083,A -85,B 0,C 180,E1 -30779.903,E2 -30779.903} C_VEL
LIN {X 0,Y 21.239,Z 462.177,A -85,B 0,C 180,E1 -30804.294,E2 -30804.294} C_VEL
LIN {X 0,Y 20.162,Z 456.874,A -85,B 0,C 180,E1 -30832.454,E2 -30832.454} C_VEL
LIN {X 0,Y 23.007,Z 450.556,A -85,B 0,C 180,E1 -30857.151,E2 -30857.151} C_VEL
LIN {X 0,Y 28.763,Z 442.564,A -85,B 0,C 180,E1 -30875.104,E2 -30875.104} C_VEL
LIN {X 0,Y 36.186,Z 432.703,A -85,B 0,C 180,E1 -30886.73,E2 -30886.73} C_VEL
LIN {X 0,Y 42.673,Z 423.172,A -85,B 0,C 180,E1 -30893.034,E2 -30893.034} C_VEL
LIN {X 0,Y 44.836,Z 419.691,A -85,B 0,C 180,E1 -30894.622,E2 -30894.622} C_VEL
LIN {X 0,Y 47.345,Z 414.753,A -85,B 0,C 180,E1 -30897.118,E2 -30897.118} C_VEL
LIN {X 0,Y 50.119,Z 406.251,A -85,B 0,C 180,E1 -30902.207,E2 -30902.207} C_VEL
LIN {X 0,Y 52.603,Z 397.465,A -85,B 0,C 180,E1 -30906.572,E2 -30906.572} C_VEL
LIN {X 0,Y 54.455,Z 391.909,A -85,B 0,C 180,E1 -30907.903,E2 -30907.903} C_VEL
LIN {X 0,Y 58.522,Z 378.82,A -85,B 0,C 180,E1 -30909.096,E2 -30909.096} C_VEL
LIN {X 0,Y 61.455,Z 364.83,A -85,B 0,C 180,E1 -30909.715,E2 -30909.715} C_VEL
LIN {X 0,Y 64.034,Z 347.441,A -85,B 0,C 180,E1 -30910.623,E2 -30910.623} C_VEL
LIN {X 0,Y 62.906,Z 342.747,A -85,B 0,C 180,E1 -30914.707,E2 -30914.707} C_VEL
LIN {X 0,Y 61.385,Z 337.098,A -85,B 0,C 180,E1 -30921.707,E2 -30921.707} C_VEL
LIN {X 0,Y 60.7,Z 335.095,A -85,B 0,C 180,E1 -30925.663,E2 -30925.663} C_VEL
LIN {X 0,Y 60.17,Z 332.799,A -85,B 0,C 180,E1 -30931.203,E2 -30931.203} C_VEL
LIN {X 0,Y 60.094,Z 332.437,A -85,B 0,C 180,E1 -30943.232,E2 -30943.232} C_VEL
LIN {X 0,Y 60.511,Z 332.911,A -85,B 0,C 180,E1 -30947.224,E2 -30947.224} C_VEL
LIN {X 0,Y 61.02,Z 335.28,A -85,B 0,C 180,E1 -30951.599,E2 -30951.599} C_VEL
LIN {X 0,Y 61.899,Z 338.951,A -85,B 0,C 180,E1 -30956.692,E2 -30956.692} C_VEL
LIN {X 0,Y 63.115,Z 344.307,A -85,B 0,C 180,E1 -30962.15,E2 -30962.15} C_VEL
LIN {X 0,Y 64.017,Z 348.966,A -85,B 0,C 180,E1 -30965.61,E2 -30965.61} C_VEL
LIN {X 0,Y 60.036,Z 373.266,A -85,B 0,C 180,E1 -30966.61,E2 -30966.61} C_VEL
LIN {X 0,Y 56.722,Z 386.01,A -85,B 0,C 180,E1 -30967.516,E2 -30967.516} C_VEL
LIN {X 0,Y 52.465,Z 397.796,A -85,B 0,C 180,E1 -30968.832,E2 -30968.832} C_VEL
LIN {X 0,Y 46.535,Z 410.189,A -85,B 0,C 180,E1 -30970.917,E2 -30970.917} C_VEL
LIN {X 0,Y 39.047,Z 422.587,A -85,B 0,C 180,E1 -30974.598,E2 -30974.598} C_VEL
LIN {X 0,Y 31.796,Z 432.517,A -85,B 0,C 180,E1 -30979.991,E2 -30979.991} C_VEL
LIN {X 0,Y 24.237,Z 441.514,A -85,B 0,C 180,E1 -30989.495,E2 -30989.495} C_VEL
LIN {X 0,Y 16.788,Z 450.272,A -85,B 0,C 180,E1 -31011.05,E2 -31011.05} C_VEL
LIN {X 0,Y 13.762,Z 457.226,A -85,B 0,C 180,E1 -31049.95,E2 -31049.95} C_VEL
LIN {X 0,Y 15.306,Z 460.947,A -85,B 0,C 180,E1 -31077.282,E2 -31077.282} C_VEL
LIN {X 0,Y 24.23,Z 466.738,A -85,B 0,C 180,E1 -31110.42,E2 -31110.42} C_VEL
LIN {X 0,Y 27.552,Z 468.068,A -85,B 0,C 180,E1 -31115.371,E2 -31115.371} C_VEL
LIN {X 0,Y 29.192,Z 468.654,A -85,B 0,C 180,E1 -31118.92,E2 -31118.92} C_VEL
LIN {X 0,Y 17.922,Z 463.312,A -85,B 0,C 180,E1 -31139.852,E2 -31139.852} C_VEL
LIN {X 0,Y 13.393,Z 458.602,A -85,B 0,C 180,E1 -31171.418,E2 -31171.418} C_VEL
LIN {X 0,Y 14.605,Z 452.424,A -85,B 0,C 180,E1 -31213.573,E2 -31213.573} C_VEL
LIN {X 0,Y 19.685,Z 446.075,A -85,B 0,C 180,E1 -31236.873,E2 -31236.873} C_VEL
LIN {X 0,Y 26.994,Z 437.749,A -85,B 0,C 180,E1 -31250.844,E2 -31250.844} C_VEL
LIN {X 0,Y 34.848,Z 427.919,A -85,B 0,C 180,E1 -31258.641,E2 -31258.641} C_VEL
LIN {X 0,Y 42.521,Z 416.55,A -85,B 0,C 180,E1 -31263.269,E2 -31263.269} C_VEL
LIN {X 0,Y 48.887,Z 404.964,A -85,B 0,C 180,E1 -31265.978,E2 -31265.978} C_VEL
LIN {X 0,Y 54.455,Z 391.909,A -85,B 0,C 180,E1 -31267.903,E2 -31267.903} C_VEL
LIN {X 0,Y 55.467,Z 388.181,A -85,B 0,C 180,E1 -31268.927,E2 -31268.927} C_VEL
LIN {X 0,Y 56.104,Z 382.198,A -85,B 0,C 180,E1 -31272.095,E2 -31272.095} C_VEL
LIN {X 0,Y 56.622,Z 376.131,A -85,B 0,C 180,E1 -31275.108,E2 -31275.108} C_VEL
LIN {X 0,Y 57.272,Z 372.267,A -85,B 0,C 180,E1 -31275.851,E2 -31275.851} C_VEL
LIN {X 0,Y 60.873,Z 350.856,A -85,B 0,C 180,E1 -31276.361,E2 -31276.361} C_VEL
LIN {X 0,Y 60.924,Z 349.855,A -85,B 0,C 180,E1 -31276.676,E2 -31276.676} C_VEL
LIN {X 0,Y 59.84,Z 344.401,A -85,B 0,C 180,E1 -31282.94,E2 -31282.94} C_VEL
LIN {X 0,Y 59.204,Z 341.593,A -85,B 0,C 180,E1 -31288.002,E2 -31288.002} C_VEL
LIN {X 0,Y 58.927,Z 339.75,A -85,B 0,C 180,E1 -31292.595,E2 -31292.595} C_VEL
LIN {X 0,Y 58.93,Z 339.428,A -85,B 0,C 180,E1 -31302.606,E2 -31302.606} C_VEL
LIN {X 0,Y 59.193,Z 339.878,A -85,B 0,C 180,E1 -31305.856,E2 -31305.856} C_VEL
LIN {X 0,Y 59.735,Z 343.599,A -85,B 0,C 180,E1 -31311.885,E2 -31311.885} C_VEL
LIN {X 0,Y 60.565,Z 348.767,A -85,B 0,C 180,E1 -31317.586,E2 -31317.586} C_VEL
LIN {X 0,Y 60.882,Z 351.174,A -85,B 0,C 180,E1 -31319.591,E2 -31319.591} C_VEL
LIN {X 0,Y 57.233,Z 373.059,A -85,B 0,C 180,E1 -31320.243,E2 -31320.243} C_VEL
LIN {X 0,Y 53.819,Z 385.853,A -85,B 0,C 180,E1 -31320.775,E2 -31320.775} C_VEL
LIN {X 0,Y 50.062,Z 396.166,A -85,B 0,C 180,E1 -31321.482,E2 -31321.482} C_VEL
LIN {X 0,Y 43.983,Z 408.891,A -85,B 0,C 180,E1 -31322.647,E2 -31322.647} C_VEL
LIN {X 0,Y 37.028,Z 420.231,A -85,B 0,C 180,E1 -31324.61,E2 -31324.61} C_VEL
LIN {X 0,Y 28.415,Z 431.534,A -85,B 0,C 180,E1 -31328.212,E2 -31328.212} C_VEL
LIN {X 0,Y 20.005,Z 440.661,A -85,B 0,C 180,E1 -31334.828,E2 -31334.828} C_VEL
LIN {X 0,Y 10.77,Z 449.502,A -85,B 0,C 180,E1 -31355.234,E2 -31355.234} C_VEL
LIN {X 0,Y 7.063,Z 456.553,A -85,B 0,C 180,E1 -31424.304,E2 -31424.304} C_VEL
LIN {X 0,Y 11.241,Z 460.554,A -85,B 0,C 180,E1 -31465.535,E2 -31465.535} C_VEL
LIN {X 0,Y 13.748,Z 461.991,A -85,B 0,C 180,E1 -31479.299,E2 -31479.299} C_VEL
LIN {X 0,Y 6.556,Z 456.757,A -85,B 0,C 180,E1 -31522.287,E2 -31522.287} C_VEL
LIN {X 0,Y 8.354,Z 451.349,A -85,B 0,C 180,E1 -31590.082,E2 -31590.082} C_VEL
LIN {X 0,Y 17.024,Z 443.193,A -85,B 0,C 180,E1 -31617.719,E2 -31617.719} C_VEL
LIN {X 0,Y 26.214,Z 433.629,A -85,B 0,C 180,E1 -31626.631,E2 -31626.631} C_VEL
LIN {X 0,Y 34.211,Z 423.731,A -85,B 0,C 180,E1 -31630.52,E2 -31630.52} C_VEL
LIN {X 0,Y 41.411,Z 412.885,A -85,B 0,C 180,E1 -31632.776,E2 -31632.776} C_VEL
LIN {X 0,Y 47.83,Z 400.704,A -85,B 0,C 180,E1 -31634.214,E2 -31634.214} C_VEL
LIN {X 0,Y 52.878,Z 388.177,A -85,B 0,C 180,E1 -31635.161,E2 -31635.161} C_VEL
LIN {X 0,Y 56.722,Z 374.682,A -85,B 0,C 180,E1 -31635.78,E2 -31635.78} C_VEL
LIN {X 0,Y 57.272,Z 372.267,A -85,B 0,C 180,E1 -31635.851,E2 -31635.851} C_VEL
LIN {X 0,Y 58.263,Z 366.761,A -85,B 0,C 180,E1 -31636.327,E2 -31636.327} C_VEL
LIN {X 0,Y 58.732,Z 361.341,A -85,B 0,C 180,E1 -31637.674,E2 -31637.674} C_VEL
LIN {X 0,Y 58.736,Z 356.431,A -85,B 0,C 180,E1 -31640.005,E2 -31640.005} C_VEL
LIN {X 0,Y 58.481,Z 353.328,A -85,B 0,C 180,E1 -31642.556,E2 -31642.556} C_VEL
LIN {X 0,Y 58.355,Z 352.474,A -85,B 0,C 180,E1 -31643.581,E2 -31643.581} C_VEL
LIN {X 0,Y 57.914,Z 348.852,A -85,B 0,C 180,E1 -31648.786,E2 -31648.786} C_VEL
LIN {X 0,Y 57.72,Z 346.618,A -85,B 0,C 180,E1 -31654.316,E2 -31654.316} C_VEL
LIN {X 0,Y 57.882,Z 346.477,A -85,B 0,C 180,E1 -31663.532,E2 -31663.532} C_VEL
LIN {X 0,Y 58.061,Z 349.912,A -85,B 0,C 180,E1 -31668.876,E2 -31668.876} C_VEL
LIN {X 0,Y 58.405,Z 353.687,A -85,B 0,C 180,E1 -31673.135,E2 -31673.135} C_VEL
LIN {X 0,Y 54.995,Z 373.435,A -85,B 0,C 180,E1 -31673.35,E2 -31673.35} C_VEL
LIN {X 0,Y 51.493,Z 386.187,A -85,B 0,C 180,E1 -31673.439,E2 -31673.439} C_VEL
LIN {X 0,Y 46.868,Z 398.254,A -85,B 0,C 180,E1 -31673.556,E2 -31673.556} C_VEL
LIN {X 0,Y 40.669,Z 410.421,A -85,B 0,C 180,E1 -31673.684,E2 -31673.684} C_VEL
LIN {X 0,Y 33.589,Z 421.404,A -85,B 0,C 180,E1 -31673.832,E2 -31673.832} C_VEL
LIN {X 0,Y 25.625,Z 431.449,A -85,B 0,C 180,E1 -31674.075,E2 -31674.075} C_VEL
LIN {X 0,Y 17.663,Z 439.74,A -85,B 0,C 180,E1 -31674.508,E2 -31674.508} C_VEL
LIN {X 0,Y 7.068,Z 448.731,A -85,B 0,C 180,E1 -31674.855,E2 -31674.855} C_VEL
LIN {X 0,Y 5.749,Z 449.718,A -85,B 0,C 180,E1 -31674.813,E2 -31674.813} C_VEL
LIN {X 0,Y 3.504,Z 451.271,A -85,B 0,C 180,E1 -31650.329,E2 -31650.329} C_VEL
LIN {X 0,Y 13.468,Z 443.416,A -85,B 0,C 180,E1 -31642.002,E2 -31642.002} C_VEL
LIN {X 0,Y 22.787,Z 434.356,A -85,B 0,C 180,E1 -31642.065,E2 -31642.065} C_VEL
LIN {X 0,Y 30.981,Z 424.675,A -85,B 0,C 180,E1 -31642.171,E2 -31642.171} C_VEL
LIN {X 0,Y 38.832,Z 413.245,A -85,B 0,C 180,E1 -31642.382,E2 -31642.382} C_VEL
LIN {X 0,Y 45.646,Z 400.521,A -85,B 0,C 180,E1 -31642.499,E2 -31642.499} C_VEL
LIN {X 0,Y 50.636,Z 388.32,A -85,B 0,C 180,E1 -31642.666,E2 -31642.666} C_VEL
LIN {X 0,Y 54.471,Z 375.195,A -85,B 0,C 180,E1 -31642.756,E2 -31642.756} C_VEL
LIN {X 0,Y 57.629,Z 358.199,A -85,B 0,C 180,E1 -31642.749,E2 -31642.749} C_VEL
LIN {X 0,Y 58.431,Z 353.076,A -85,B 0,C 180,E1 -31642.894,E2 -31642.894} C_VEL
LIN {X 0,Y 58.355,Z 352.474,A -85,B 0,C 180,E1 -31643.581,E2 -31643.581} C_VEL
LIN {X 0,Y 57.946,Z 351.029,A -85,B 0,C 180,E1 -31646.556,E2 -31646.556} C_VEL
LIN {X 0,Y 57.346,Z 350.512,A -85,B 0,C 180,E1 -31651.248,E2 -31651.248} C_VEL
LIN {X 0,Y 56.866,Z 351.55,A -85,B 0,C 180,E1 -31656.809,E2 -31656.809} C_VEL
LIN {X 0,Y 56.607,Z 353.864,A -85,B 0,C 180,E1 -31662.179,E2 -31662.179} C_VEL
LIN {X 0,Y 56.564,Z 355.426,A -85,B 0,C 180,E1 -31664.66,E2 -31664.66} C_VEL
LIN {X 0,Y 56.559,Z 356.537,A -85,B 0,C 180,E1 -31666.117,E2 -31666.117} C_VEL
LIN {X 0,Y 54.061,Z 371.392,A -85,B 0,C 180,E1 -31666.042,E2 -31666.042} C_VEL
LIN {X 0,Y 50.966,Z 383.551,A -85,B 0,C 180,E1 -31665.662,E2 -31665.662} C_VEL
LIN {X 0,Y 46.39,Z 396.171,A -85,B 0,C 180,E1 -31665.027,E2 -31665.027} C_VEL
LIN {X 0,Y 40.269,Z 408.851,A -85,B 0,C 180,E1 -31663.776,E2 -31663.776} C_VEL
LIN {X 0,Y 33.291,Z 420.107,A -85,B 0,C 180,E1 -31661.868,E2 -31661.868} C_VEL
LIN {X 0,Y 28.403,Z 426.796,A -85,B 0,C 180,E1 -31659.917,E2 -31659.917} C_VEL
LIN {X 0,Y 27.074,Z 428.463,A -85,B 0,C 180,E1 -31656.922,E2 -31656.922} C_VEL
LIN {X 0,Y 34.3,Z 418.599,A -85,B 0,C 180,E1 -31653.988,E2 -31653.988} C_VEL
LIN {X 0,Y 40.965,Z 407.442,A -85,B 0,C 180,E1 -31652.117,E2 -31652.117} C_VEL
LIN {X 0,Y 46.799,Z 395.03,A -85,B 0,C 180,E1 -31651.053,E2 -31651.053} C_VEL
LIN {X 0,Y 51.407,Z 381.87,A -85,B 0,C 180,E1 -31650.426,E2 -31650.426} C_VEL
LIN {X 0,Y 54.779,Z 367.301,A -85,B 0,C 180,E1 -31649.949,E2 -31649.949} C_VEL
LIN {X 0,Y 56.56,Z 356.34,A -85,B 0,C 180,E1 -31649.902,E2 -31649.902} C_VEL
LIN {X 0,Y 56.533,Z 354.439,A -85,B 0,C 180,E1 -31653.339,E2 -31653.339} C_VEL
LIN {X 0,Y 56.554,Z 353.564,A -85,B 0,C 180,E1 -31656.129,E2 -31656.129} C_VEL
LIN {X 0,Y 56.626,Z 353.647,A -85,B 0,C 180,E1 -31661.998,E2 -31661.998} C_VEL
LIN {X 0,Y 56.564,Z 355.426,A -85,B 0,C 180,E1 -31664.66,E2 -31664.66} C_VEL
LIN {X 0,Y 56.431,Z 357.602,A -85,B 0,C 180,E1 -31666.387,E2 -31666.387} C_VEL
LIN {X 0,Y 55.993,Z 361.149,A -85,B 0,C 180,E1 -31667.218,E2 -31667.218} C_VEL
LIN {X 0,Y 55.065,Z 366.342,A -85,B 0,C 180,E1 -31666.699,E2 -31666.699} C_VEL
LIN {X 0,Y 54.034,Z 370.924,A -85,B 0,C 180,E1 -31665.078,E2 -31665.078} C_VEL
LIN {X 0,Y 53.107,Z 374.248,A -85,B 0,C 180,E1 -31662.511,E2 -31662.511} C_VEL
LIN {X 0,Y 52.694,Z 375.545,A -85,B 0,C 180,E1 -31659.826,E2 -31659.826} C_VEL
LIN {X 0,Y 52.703,Z 375.425,A -85,B 0,C 180,E1 -31658.295,E2 -31658.295} C_VEL
LIN {X 0,Y 52.74,Z 375.269,A -85,B 0,C 180,E1 -31657.908,E2 -31657.908} C_VEL
LIN {X 0,Y 55.433,Z 360.562,A -85,B 0,C 180,E1 -31657.151,E2 -31657.151} C_VEL
LIN {X 0,Y 55.438,Z 360.477,A -85,B 0,C 180,E1 -31658.927,E2 -31658.927} C_VEL
LIN {X 0,Y 52.703,Z 375.425,A -85,B 0,C 180,E1 -31658.295,E2 -31658.295} C_VEL
LIN {X 0,Y 52.654,Z 375.871,A -85,B 0,C 180,E1 -31658.285,E2 -31658.285} C_VEL
LIN {X 0,Y 52.654,Z 600,A -85,B 0,C 180,E1 -31658.285,E2 -31658.285} C_VEL
LIN {X 0,Y 52.654,Z 600,A -85,B 0,C 180,E1 -31658.285,E2 -31658.285}

QRS_NEXT_CUT()

QRS_NEXT()
QRS_HOME()

END
